LIN {X -0.159,Y -467.069,Z 497.488,A 0.000,B 0.000,C 90.000,E1 267.879} C_DIS
LIN {X -0.213,Y -463.902,Z 497.487,A 0.000,B 0.000,C 90.000,E1 267.650} C_DIS
LIN {X 0.193,Y -457.241,Z 497.485,A 0.000,B 0.000,C 90.000,E1 267.192} C_DIS
LIN {X -0.207,Y -450.486,Z 497.483,A 0.000,B 0.000,C 90.000,E1 266.906} C_DIS
LIN {X -0.134,Y -443.636,Z 497.481,A 0.000,B 0.000,C 90.000,E1 266.617} C_DIS
LIN {X -0.213,Y -436.403,Z 497.480,A 0.000,B 0.000,C 90.000,E1 266.388} C_DIS
LIN {X 0.056,Y -428.030,Z 497.479,A 0.000,B 0.000,C 90.000,E1 266.159} C_DIS
LIN {X -0.086,Y -418.559,Z 497.478,A 0.000,B 0.000,C 90.000,E1 266.045} C_DIS
LIN {X -0.068,Y -410.848,Z 497.478,A 0.000,B 0.000,C 90.000,E1 265.988} C_DIS
LIN {X -0.145,Y -404.938,Z 497.478,A 0.000,B 0.000,C 90.000,E1 265.988} C_DIS
LIN {X 0.081,Y -180.918,Z 497.478,A 0.000,B 0.000,C 90.000,E1 265.931} C_DIS
LIN {X -0.058,Y -180.845,Z 497.472,A 0.000,B 0.000,C 90.000,E1 264.951} C_DIS
LIN {X 0.019,Y -178.890,Z 497.443,A 0.000,B 0.000,C 90.000,E1 259.690} C_DIS
LIN {X -0.077,Y -175.932,Z 497.414,A 0.000,B 0.000,C 90.000,E1 254.629} C_DIS
LIN {X 0.040,Y -175.379,Z 497.410,A 0.000,B 0.000,C 90.000,E1 253.740} C_DIS
LIN {X 0.037,Y -172.153,Z 497.386,A 0.000,B 0.000,C 90.000,E1 249.464} C_DIS
LIN {X 0.074,Y -171.618,Z 497.381,A 0.000,B 0.000,C 90.000,E1 248.592} C_DIS
LIN {X 0.062,Y -167.841,Z 497.357,A 0.000,B 0.000,C 90.000,E1 244.280} C_DIS
LIN {X 0.002,Y -166.570,Z 497.348,A 0.000,B 0.000,C 90.000,E1 242.564} C_DIS
LIN {X -0.012,Y -162.563,Z 497.323,A 0.000,B 0.000,C 90.000,E1 238.201} C_DIS
LIN {X 0.048,Y -161.244,Z 497.314,A 0.000,B 0.000,C 90.000,E1 236.421} C_DIS
LIN {X -0.041,Y -157.247,Z 497.289,A 0.000,B 0.000,C 90.000,E1 232.029} C_DIS
LIN {X 0.005,Y -155.969,Z 497.279,A 0.000,B 0.000,C 90.000,E1 230.231} C_DIS
LIN {X 0.063,Y -152.224,Z 497.254,A 0.000,B 0.000,C 90.000,E1 225.729} C_DIS
LIN {X -0.027,Y -150.467,Z 497.239,A 0.000,B 0.000,C 90.000,E1 223.056} C_DIS
LIN {X -0.006,Y -147.192,Z 497.214,A 0.000,B 0.000,C 90.000,E1 218.508} C_DIS
LIN {X 0.076,Y -145.211,Z 497.194,A 0.000,B 0.000,C 90.000,E1 214.818} C_DIS
LIN {X -0.015,Y -142.344,Z 497.163,A 0.000,B 0.000,C 90.000,E1 209.333} C_DIS
LIN {X 0.039,Y -141.732,Z 497.153,A 0.000,B 0.000,C 90.000,E1 207.462} C_DIS
LIN {X 0.020,Y -139.483,Z 497.117,A 0.000,B 0.000,C 90.000,E1 200.972} C_DIS
LIN {X 0.009,Y -138.982,Z 497.101,A 0.000,B 0.000,C 90.000,E1 198.181} C_DIS
LIN {X -0.030,Y -138.333,Z 497.054,A 0.000,B 0.000,C 90.000,E1 189.792} C_DIS
LIN {X -0.006,Y -139.426,Z 497.008,A 0.000,B 0.000,C 90.000,E1 181.375} C_DIS
LIN {X 0.048,Y -141.349,Z 496.971,A 0.000,B 0.000,C 90.000,E1 174.837} C_DIS
LIN {X 0.025,Y -142.704,Z 496.956,A 0.000,B 0.000,C 90.000,E1 172.064} C_DIS
LIN {X -0.017,Y -145.075,Z 496.930,A 0.000,B 0.000,C 90.000,E1 167.465} C_DIS
LIN {X -0.020,Y -147.700,Z 496.910,A 0.000,B 0.000,C 90.000,E1 163.795} C_DIS
LIN {X 0.013,Y -150.352,Z 496.890,A 0.000,B 0.000,C 90.000,E1 160.134} C_DIS
LIN {X 0.005,Y -154.606,Z 496.865,A 0.000,B 0.000,C 90.000,E1 155.613} C_DIS
LIN {X 0.012,Y -158.148,Z 496.845,A 0.000,B 0.000,C 90.000,E1 152.025} C_DIS
LIN {X 0.057,Y -162.434,Z 496.825,A 0.000,B 0.000,C 90.000,E1 148.456} C_DIS
LIN {X -0.048,Y -166.694,Z 496.805,A 0.000,B 0.000,C 90.000,E1 144.975} C_DIS
LIN {X 0.066,Y -171.699,Z 496.786,A 0.000,B 0.000,C 90.000,E1 141.457} C_DIS
LIN {X 0.001,Y -176.673,Z 496.767,A 0.000,B 0.000,C 90.000,E1 138.038} C_DIS
LIN {X -0.006,Y -180.969,Z 496.753,A 0.000,B 0.000,C 90.000,E1 135.486} C_DIS
LIN {X -0.018,Y -186.393,Z 496.734,A 0.000,B 0.000,C 90.000,E1 132.123} C_DIS
LIN {X -0.078,Y -191.022,Z 496.720,A 0.000,B 0.000,C 90.000,E1 129.644} C_DIS
LIN {X -0.011,Y -192.947,Z 496.714,A 0.000,B 0.000,C 90.000,E1 128.463} C_DIS
LIN {X -0.063,Y -289.891,Z 496.714,A 0.000,B 0.000,C 90.000,E1 128.463} C_DIS
LIN {X -0.037,Y -294.322,Z 496.713,A 0.000,B 0.000,C 90.000,E1 128.338} C_DIS
LIN {X -0.058,Y -296.327,Z 496.712,A 0.000,B 0.000,C 90.000,E1 128.222} C_DIS
LIN {X -0.001,Y -299.079,Z 496.711,A 0.000,B 0.000,C 90.000,E1 127.971} C_DIS
LIN {X 0.099,Y -302.846,Z 496.708,A 0.000,B 0.000,C 90.000,E1 127.443} C_DIS
LIN {X -0.139,Y -304.561,Z 496.706,A 0.000,B 0.000,C 90.000,E1 127.156} C_DIS
LIN {X 0.049,Y -305.909,Z 496.704,A 0.000,B 0.000,C 90.000,E1 126.790} C_DIS
LIN {X 0.014,Y -317.009,Z 496.685,A 0.000,B 0.000,C 90.000,E1 123.214} C_DIS
LIN {X 0.034,Y -327.372,Z 496.669,A 0.000,B 0.000,C 90.000,E1 120.335} C_DIS
LIN {X 0.035,Y -339.088,Z 496.653,A 0.000,B 0.000,C 90.000,E1 117.513} C_DIS
LIN {X -0.109,Y -352.268,Z 496.638,A 0.000,B 0.000,C 90.000,E1 114.771} C_DIS
LIN {X 0.090,Y -365.305,Z 496.624,A 0.000,B 0.000,C 90.000,E1 112.333} C_DIS
LIN {X 0.000,Y -379.685,Z 496.611,A 0.000,B 0.000,C 90.000,E1 109.993} C_DIS
LIN {X 0.004,Y -395.513,Z 496.598,A 0.000,B 0.000,C 90.000,E1 107.692} C_DIS
LIN {X 0.171,Y -412.905,Z 496.586,A 0.000,B 0.000,C 90.000,E1 105.426} C_DIS
LIN {X 0.169,Y -431.991,Z 496.574,A 0.000,B 0.000,C 90.000,E1 103.244} C_DIS
LIN {X -0.185,Y -452.129,Z 496.562,A 0.000,B 0.000,C 90.000,E1 101.243} C_DIS
LIN {X 0.176,Y -472.814,Z 496.552,A 0.000,B 0.000,C 90.000,E1 99.321} C_DIS
LIN {X -0.004,Y -480.554,Z 496.548,A 0.000,B 0.000,C 90.000,E1 98.681} C_DIS
LIN {X 0.071,Y -482.476,Z 496.547,A 0.000,B 0.000,C 90.000,E1 98.454} C_DIS
LIN {X -0.051,Y -484.150,Z 496.546,A 0.000,B 0.000,C 90.000,E1 98.219} C_DIS
LIN {X -0.242,Y -485.406,Z 496.544,A 0.000,B 0.000,C 90.000,E1 97.992} C_DIS
LIN {X 0.010,Y -486.954,Z 496.541,A 0.000,B 0.000,C 90.000,E1 97.466} C_DIS
LIN {X 0.203,Y -487.446,Z 496.539,A 0.000,B 0.000,C 90.000,E1 96.947} C_DIS
LIN {X -0.078,Y -486.959,Z 496.536,A 0.000,B 0.000,C 90.000,E1 96.486} C_DIS
LIN {X 0.128,Y -485.415,Z 496.533,A 0.000,B 0.000,C 90.000,E1 95.967} C_DIS
LIN {X -0.037,Y -484.162,Z 496.532,A 0.000,B 0.000,C 90.000,E1 95.739} C_DIS
LIN {X -0.199,Y -482.489,Z 496.530,A 0.000,B 0.000,C 90.000,E1 95.511} C_DIS
LIN {X 0.089,Y -468.245,Z 496.521,A 0.000,B 0.000,C 90.000,E1 93.726} C_DIS
LIN {X 0.037,Y -455.064,Z 496.511,A 0.000,B 0.000,C 90.000,E1 91.949} C_DIS
LIN {X 0.020,Y -436.764,Z 496.495,A 0.000,B 0.000,C 90.000,E1 89.083} C_DIS
LIN {X -0.075,Y -423.680,Z 496.483,A 0.000,B 0.000,C 90.000,E1 86.963} C_DIS
LIN {X -0.085,Y -412.501,Z 496.473,A 0.000,B 0.000,C 90.000,E1 85.065} C_DIS
LIN {X -0.194,Y -398.290,Z 496.459,A 0.000,B 0.000,C 90.000,E1 82.591} C_DIS
LIN {X 0.156,Y -387.289,Z 496.448,A 0.000,B 0.000,C 90.000,E1 80.566} C_DIS
LIN {X 0.036,Y -374.741,Z 496.435,A 0.000,B 0.000,C 90.000,E1 78.285} C_DIS
LIN {X 0.008,Y -359.680,Z 496.419,A 0.000,B 0.000,C 90.000,E1 75.353} C_DIS
LIN {X -0.041,Y -349.044,Z 496.405,A 0.000,B 0.000,C 90.000,E1 72.960} C_DIS
LIN {X 0.086,Y -335.271,Z 496.385,A 0.000,B 0.000,C 90.000,E1 69.263} C_DIS
LIN {X -0.128,Y -324.859,Z 496.368,A 0.000,B 0.000,C 90.000,E1 66.177} C_DIS
LIN {X -0.128,Y -316.777,Z 496.353,A 0.000,B 0.000,C 90.000,E1 63.640} C_DIS
LIN {X -0.043,Y -308.825,Z 496.339,A 0.000,B 0.000,C 90.000,E1 61.051} C_DIS
LIN {X -0.122,Y -300.916,Z 496.325,A 0.000,B 0.000,C 90.000,E1 58.456} C_DIS
LIN {X 0.082,Y -291.407,Z 496.306,A 0.000,B 0.000,C 90.000,E1 55.102} C_DIS
LIN {X -0.032,Y -284.211,Z 496.291,A 0.000,B 0.000,C 90.000,E1 52.431} C_DIS
LIN {X 0.125,Y -278.713,Z 496.280,A 0.000,B 0.000,C 90.000,E1 50.356} C_DIS
LIN {X -0.028,Y -274.824,Z 496.272,A 0.000,B 0.000,C 90.000,E1 49.013} C_DIS
LIN {X -0.048,Y -270.703,Z 496.265,A 0.000,B 0.000,C 90.000,E1 47.634} C_DIS
LIN {X 0.005,Y -264.053,Z 496.253,A 0.000,B 0.000,C 90.000,E1 45.526} C_DIS
LIN {X -0.062,Y -255.999,Z 496.239,A 0.000,B 0.000,C 90.000,E1 43.056} C_DIS
LIN {X -0.069,Y -245.974,Z 496.221,A 0.000,B 0.000,C 90.000,E1 39.806} C_DIS
LIN {X 0.062,Y -235.445,Z 496.201,A 0.000,B 0.000,C 90.000,E1 36.091} C_DIS
LIN {X 0.070,Y -227.752,Z 496.184,A 0.000,B 0.000,C 90.000,E1 33.086} C_DIS
LIN {X 0.016,Y -221.019,Z 496.167,A 0.000,B 0.000,C 90.000,E1 30.050} C_DIS
LIN {X 0.048,Y -215.087,Z 496.150,A 0.000,B 0.000,C 90.000,E1 26.950} C_DIS
LIN {X 0.033,Y -210.049,Z 496.132,A 0.000,B 0.000,C 90.000,E1 23.823} C_DIS
LIN {X -0.045,Y -204.859,Z 496.110,A 0.000,B 0.000,C 90.000,E1 19.885} C_DIS
LIN {X 0.094,Y -200.523,Z 496.088,A 0.000,B 0.000,C 90.000,E1 15.843} C_DIS
LIN {X 0.044,Y -196.735,Z 496.061,A 0.000,B 0.000,C 90.000,E1 11.007} C_DIS
LIN {X 0.081,Y -193.879,Z 496.025,A 0.000,B 0.000,C 90.000,E1 4.473} C_DIS
LIN {X -0.057,Y -194.901,Z 495.961,A 0.000,B 0.000,C 90.000,E1 352.996} C_DIS
LIN {X -0.067,Y -197.808,Z 495.934,A 0.000,B 0.000,C 90.000,E1 348.105} C_DIS
LIN {X 0.014,Y -201.345,Z 495.911,A 0.000,B 0.000,C 90.000,E1 344.031} C_DIS
LIN {X 0.035,Y -205.757,Z 495.889,A 0.000,B 0.000,C 90.000,E1 340.007} C_DIS
LIN {X -0.038,Y -211.033,Z 495.867,A 0.000,B 0.000,C 90.000,E1 336.049} C_DIS
LIN {X 0.016,Y -216.916,Z 495.845,A 0.000,B 0.000,C 90.000,E1 332.103} C_DIS
LIN {X 0.093,Y -223.417,Z 495.823,A 0.000,B 0.000,C 90.000,E1 328.201} C_DIS
LIN {X -0.023,Y -230.541,Z 495.802,A 0.000,B 0.000,C 90.000,E1 324.402} C_DIS
LIN {X -0.069,Y -238.308,Z 495.781,A 0.000,B 0.000,C 90.000,E1 320.642} C_DIS
LIN {X 0.042,Y -247.097,Z 495.761,A 0.000,B 0.000,C 90.000,E1 316.905} C_DIS
LIN {X 0.028,Y -253.961,Z 495.746,A 0.000,B 0.000,C 90.000,E1 314.352} C_DIS
LIN {X -0.044,Y -264.868,Z 495.727,A 0.000,B 0.000,C 90.000,E1 310.782} C_DIS
LIN {X 0.031,Y -275.649,Z 495.709,A 0.000,B 0.000,C 90.000,E1 307.604} C_DIS
LIN {X -0.123,Y -288.837,Z 495.690,A 0.000,B 0.000,C 90.000,E1 304.199} C_DIS
LIN {X 0.128,Y -301.582,Z 495.673,A 0.000,B 0.000,C 90.000,E1 301.131} C_DIS
LIN {X -0.084,Y -316.818,Z 495.655,A 0.000,B 0.000,C 90.000,E1 297.897} C_DIS
LIN {X -0.042,Y -330.447,Z 495.641,A 0.000,B 0.000,C 90.000,E1 295.335} C_DIS
LIN {X 0.069,Y -343.666,Z 495.629,A 0.000,B 0.000,C 90.000,E1 293.131} C_DIS
LIN {X 0.220,Y -358.136,Z 495.617,A 0.000,B 0.000,C 90.000,E1 290.972} C_DIS
LIN {X 0.100,Y -373.737,Z 495.605,A 0.000,B 0.000,C 90.000,E1 288.906} C_DIS
LIN {X -0.133,Y -393.034,Z 495.592,A 0.000,B 0.000,C 90.000,E1 286.622} C_DIS
LIN {X -0.119,Y -415.555,Z 495.578,A 0.000,B 0.000,C 90.000,E1 284.120} C_DIS
LIN {X -0.049,Y -428.141,Z 495.571,A 0.000,B 0.000,C 90.000,E1 282.771} C_DIS
LIN {X 0.056,Y -440.413,Z 495.564,A 0.000,B 0.000,C 90.000,E1 281.422} C_DIS
LIN {X 0.058,Y -449.879,Z 495.558,A 0.000,B 0.000,C 90.000,E1 280.366} C_DIS
LIN {X -0.177,Y -456.408,Z 495.553,A 0.000,B 0.000,C 90.000,E1 279.613} C_DIS
LIN {X 0.106,Y -462.355,Z 495.549,A 0.000,B 0.000,C 90.000,E1 278.803} C_DIS
LIN {X -0.018,Y -467.762,Z 495.545,A 0.000,B 0.000,C 90.000,E1 278.049} C_DIS
LIN {X -0.092,Y -472.644,Z 495.540,A 0.000,B 0.000,C 90.000,E1 277.296} C_DIS
LIN {X -0.133,Y -476.909,Z 495.536,A 0.000,B 0.000,C 90.000,E1 276.543} C_DIS
LIN {X -0.187,Y -480.642,Z 495.532,A 0.000,B 0.000,C 90.000,E1 275.796} C_DIS
LIN {X -0.209,Y -483.765,Z 495.528,A 0.000,B 0.000,C 90.000,E1 275.049} C_DIS
LIN {X -0.037,Y -485.507,Z 495.525,A 0.000,B 0.000,C 90.000,E1 274.531} C_DIS
LIN {X 0.145,Y -486.903,Z 495.522,A 0.000,B 0.000,C 90.000,E1 274.012} C_DIS
LIN {X -0.182,Y -487.979,Z 495.520,A 0.000,B 0.000,C 90.000,E1 273.555} C_DIS
LIN {X 0.016,Y -488.764,Z 495.517,A 0.000,B 0.000,C 90.000,E1 273.037} C_DIS
LIN {X 0.194,Y -489.189,Z 495.514,A 0.000,B 0.000,C 90.000,E1 272.522} C_DIS
LIN {X -0.109,Y -489.235,Z 495.511,A 0.000,B 0.000,C 90.000,E1 272.064} C_DIS
LIN {X 0.095,Y -488.877,Z 495.509,A 0.000,B 0.000,C 90.000,E1 271.547} C_DIS
LIN {X -0.204,Y -488.107,Z 495.506,A 0.000,B 0.000,C 90.000,E1 271.088} C_DIS
LIN {X -0.016,Y -486.833,Z 495.503,A 0.000,B 0.000,C 90.000,E1 270.573} C_DIS
LIN {X 0.167,Y -485.001,Z 495.500,A 0.000,B 0.000,C 90.000,E1 270.057} C_DIS
LIN {X -0.141,Y -482.512,Z 495.498,A 0.000,B 0.000,C 90.000,E1 269.599} C_DIS
LIN {X 0.017,Y -479.232,Z 495.495,A 0.000,B 0.000,C 90.000,E1 269.083} C_DIS
LIN {X 0.155,Y -475.095,Z 495.492,A 0.000,B 0.000,C 90.000,E1 268.568} C_DIS
LIN {X -0.025,Y -472.680,Z 495.491,A 0.000,B 0.000,C 90.000,E1 268.339} C_DIS
LIN {X -0.224,Y -467.092,Z 495.488,A 0.000,B 0.000,C 90.000,E1 267.879} C_DIS
LIN {X -0.049,Y -460.845,Z 495.486,A 0.000,B 0.000,C 90.000,E1 267.421} C_DIS
LIN {X 0.179,Y -454.124,Z 495.484,A 0.000,B 0.000,C 90.000,E1 267.020} C_DIS
LIN {X 0.007,Y -447.262,Z 495.482,A 0.000,B 0.000,C 90.000,E1 266.731} C_DIS
LIN {X 0.211,Y -440.273,Z 495.480,A 0.000,B 0.000,C 90.000,E1 266.445} C_DIS
LIN {X -0.102,Y -432.652,Z 495.479,A 0.000,B 0.000,C 90.000,E1 266.274} C_DIS
LIN {X -0.021,Y -424.203,Z 495.478,A 0.000,B 0.000,C 90.000,E1 266.102} C_DIS
LIN {X 0.001,Y -413.442,Z 495.478,A 0.000,B 0.000,C 90.000,E1 265.988} C_DIS
LIN {X -0.161,Y -406.443,Z 495.478,A 0.000,B 0.000,C 90.000,E1 265.988} C_DIS
LIN {X 0.073,Y -180.918,Z 495.478,A 0.000,B 0.000,C 90.000,E1 265.931} C_DIS
LIN {X -0.068,Y -180.845,Z 495.472,A 0.000,B 0.000,C 90.000,E1 264.951} C_DIS
LIN {X 0.008,Y -178.889,Z 495.443,A 0.000,B 0.000,C 90.000,E1 259.690} C_DIS
LIN {X 0.083,Y -175.931,Z 495.414,A 0.000,B 0.000,C 90.000,E1 254.574} C_DIS
LIN {X 0.029,Y -175.376,Z 495.410,A 0.000,B 0.000,C 90.000,E1 253.740} C_DIS
LIN {X 0.027,Y -172.151,Z 495.386,A 0.000,B 0.000,C 90.000,E1 249.464} C_DIS
LIN {X 0.065,Y -171.617,Z 495.381,A 0.000,B 0.000,C 90.000,E1 248.592} C_DIS
LIN {X 0.053,Y -167.839,Z 495.357,A 0.000,B 0.000,C 90.000,E1 244.280} C_DIS
LIN {X -0.007,Y -166.567,Z 495.348,A 0.000,B 0.000,C 90.000,E1 242.564} C_DIS
LIN {X -0.020,Y -162.561,Z 495.323,A 0.000,B 0.000,C 90.000,E1 238.201} C_DIS
LIN {X 0.039,Y -161.240,Z 495.314,A 0.000,B 0.000,C 90.000,E1 236.421} C_DIS
LIN {X 0.074,Y -157.244,Z 495.289,A 0.000,B 0.000,C 90.000,E1 231.984} C_DIS
LIN {X -0.004,Y -155.967,Z 495.279,A 0.000,B 0.000,C 90.000,E1 230.231} C_DIS
LIN {X 0.054,Y -152.222,Z 495.254,A 0.000,B 0.000,C 90.000,E1 225.729} C_DIS
LIN {X -0.035,Y -150.465,Z 495.239,A 0.000,B 0.000,C 90.000,E1 223.056} C_DIS
LIN {X -0.015,Y -147.190,Z 495.214,A 0.000,B 0.000,C 90.000,E1 218.508} C_DIS
LIN {X 0.067,Y -145.209,Z 495.194,A 0.000,B 0.000,C 90.000,E1 214.818} C_DIS
LIN {X -0.023,Y -142.343,Z 495.163,A 0.000,B 0.000,C 90.000,E1 209.333} C_DIS
LIN {X 0.030,Y -141.731,Z 495.153,A 0.000,B 0.000,C 90.000,E1 207.462} C_DIS
LIN {X 0.012,Y -139.483,Z 495.117,A 0.000,B 0.000,C 90.000,E1 200.972} C_DIS
LIN {X 0.000,Y -138.982,Z 495.101,A 0.000,B 0.000,C 90.000,E1 198.181} C_DIS
LIN {X -0.038,Y -138.333,Z 495.054,A 0.000,B 0.000,C 90.000,E1 189.792} C_DIS
LIN {X -0.014,Y -139.427,Z 495.008,A 0.000,B 0.000,C 90.000,E1 181.375} C_DIS
LIN {X 0.040,Y -141.351,Z 494.971,A 0.000,B 0.000,C 90.000,E1 174.837} C_DIS
LIN {X 0.016,Y -142.705,Z 494.956,A 0.000,B 0.000,C 90.000,E1 172.064} C_DIS
LIN {X -0.025,Y -145.077,Z 494.930,A 0.000,B 0.000,C 90.000,E1 167.465} C_DIS
LIN {X -0.029,Y -147.702,Z 494.910,A 0.000,B 0.000,C 90.000,E1 163.795} C_DIS
LIN {X 0.054,Y -150.355,Z 494.890,A 0.000,B 0.000,C 90.000,E1 160.115} C_DIS
LIN {X 0.073,Y -153.779,Z 494.870,A 0.000,B 0.000,C 90.000,E1 156.485} C_DIS
LIN {X -0.007,Y -157.191,Z 494.850,A 0.000,B 0.000,C 90.000,E1 152.922} C_DIS
LIN {X 0.076,Y -161.351,Z 494.830,A 0.000,B 0.000,C 90.000,E1 149.331} C_DIS
LIN {X 0.088,Y -165.554,Z 494.810,A 0.000,B 0.000,C 90.000,E1 145.801} C_DIS
LIN {X -0.028,Y -170.468,Z 494.791,A 0.000,B 0.000,C 90.000,E1 142.351} C_DIS
LIN {X -0.011,Y -175.350,Z 494.772,A 0.000,B 0.000,C 90.000,E1 138.895} C_DIS
LIN {X -0.015,Y -180.974,Z 494.753,A 0.000,B 0.000,C 90.000,E1 135.486} C_DIS
LIN {X -0.028,Y -186.398,Z 494.734,A 0.000,B 0.000,C 90.000,E1 132.123} C_DIS
LIN {X -0.088,Y -191.027,Z 494.720,A 0.000,B 0.000,C 90.000,E1 129.644} C_DIS
LIN {X 0.094,Y -193.031,Z 494.713,A 0.000,B 0.000,C 90.000,E1 128.382} C_DIS
LIN {X 0.097,Y -290.712,Z 494.713,A 0.000,B 0.000,C 90.000,E1 128.382} C_DIS
LIN {X 0.009,Y -291.718,Z 494.713,A 0.000,B 0.000,C 90.000,E1 128.382} C_DIS
LIN {X -0.005,Y -296.314,Z 494.712,A 0.000,B 0.000,C 90.000,E1 128.177} C_DIS
LIN {X -0.017,Y -298.790,Z 494.711,A 0.000,B 0.000,C 90.000,E1 127.971} C_DIS
LIN {X 0.163,Y -302.616,Z 494.708,A 0.000,B 0.000,C 90.000,E1 127.443} C_DIS
LIN {X -0.075,Y -304.406,Z 494.706,A 0.000,B 0.000,C 90.000,E1 127.156} C_DIS
LIN {X 0.111,Y -305.809,Z 494.704,A 0.000,B 0.000,C 90.000,E1 126.790} C_DIS
LIN {X -0.089,Y -307.846,Z 494.701,A 0.000,B 0.000,C 90.000,E1 126.171} C_DIS
LIN {X 0.148,Y -318.034,Z 494.683,A 0.000,B 0.000,C 90.000,E1 122.880} C_DIS
LIN {X -0.076,Y -328.534,Z 494.667,A 0.000,B 0.000,C 90.000,E1 120.050} C_DIS
LIN {X 0.086,Y -340.403,Z 494.651,A 0.000,B 0.000,C 90.000,E1 117.206} C_DIS
LIN {X -0.006,Y -353.742,Z 494.636,A 0.000,B 0.000,C 90.000,E1 114.463} C_DIS
LIN {X -0.103,Y -366.936,Z 494.623,A 0.000,B 0.000,C 90.000,E1 112.078} C_DIS
LIN {X 0.065,Y -381.483,Z 494.610,A 0.000,B 0.000,C 90.000,E1 109.704} C_DIS
LIN {X 0.127,Y -397.492,Z 494.597,A 0.000,B 0.000,C 90.000,E1 107.402} C_DIS
LIN {X -0.040,Y -415.080,Z 494.584,A 0.000,B 0.000,C 90.000,E1 105.190} C_DIS
LIN {X 0.030,Y -434.343,Z 494.572,A 0.000,B 0.000,C 90.000,E1 103.008} C_DIS
LIN {X -0.167,Y -454.551,Z 494.561,A 0.000,B 0.000,C 90.000,E1 101.007} C_DIS
LIN {X -0.193,Y -475.297,Z 494.551,A 0.000,B 0.000,C 90.000,E1 99.151} C_DIS
LIN {X 0.060,Y -480.475,Z 494.548,A 0.000,B 0.000,C 90.000,E1 98.681} C_DIS
LIN {X 0.135,Y -482.460,Z 494.547,A 0.000,B 0.000,C 90.000,E1 98.454} C_DIS
LIN {X 0.013,Y -484.182,Z 494.546,A 0.000,B 0.000,C 90.000,E1 98.219} C_DIS
LIN {X -0.178,Y -485.476,Z 494.544,A 0.000,B 0.000,C 90.000,E1 97.992} C_DIS
LIN {X 0.074,Y -487.079,Z 494.542,A 0.000,B 0.000,C 90.000,E1 97.466} C_DIS
LIN {X -0.216,Y -487.616,Z 494.539,A 0.000,B 0.000,C 90.000,E1 97.004} C_DIS
LIN {X -0.013,Y -487.173,Z 494.536,A 0.000,B 0.000,C 90.000,E1 96.486} C_DIS
LIN {X 0.193,Y -485.682,Z 494.533,A 0.000,B 0.000,C 90.000,E1 95.967} C_DIS
LIN {X 0.030,Y -484.462,Z 494.532,A 0.000,B 0.000,C 90.000,E1 95.739} C_DIS
LIN {X -0.132,Y -482.833,Z 494.531,A 0.000,B 0.000,C 90.000,E1 95.511} C_DIS
LIN {X -0.114,Y -470.618,Z 494.522,A 0.000,B 0.000,C 90.000,E1 94.012} C_DIS
LIN {X -0.125,Y -457.192,Z 494.512,A 0.000,B 0.000,C 90.000,E1 92.236} C_DIS
LIN {X 0.066,Y -445.210,Z 494.502,A 0.000,B 0.000,C 90.000,E1 90.401} C_DIS
LIN {X -0.002,Y -433.770,Z 494.492,A 0.000,B 0.000,C 90.000,E1 88.568} C_DIS
LIN {X 0.100,Y -417.547,Z 494.477,A 0.000,B 0.000,C 90.000,E1 85.869} C_DIS
LIN {X 0.028,Y -404.810,Z 494.465,A 0.000,B 0.000,C 90.000,E1 83.685} C_DIS
LIN {X 0.074,Y -393.852,Z 494.454,A 0.000,B 0.000,C 90.000,E1 81.724} C_DIS
LIN {X 0.002,Y -382.829,Z 494.443,A 0.000,B 0.000,C 90.000,E1 79.746} C_DIS
LIN {X 0.152,Y -370.337,Z 494.430,A 0.000,B 0.000,C 90.000,E1 77.409} C_DIS
LIN {X 0.111,Y -359.905,Z 494.419,A 0.000,B 0.000,C 90.000,E1 75.353} C_DIS
LIN {X -0.013,Y -348.012,Z 494.404,A 0.000,B 0.000,C 90.000,E1 72.670} C_DIS
LIN {X 0.193,Y -335.424,Z 494.385,A 0.000,B 0.000,C 90.000,E1 69.263} C_DIS
LIN {X -0.020,Y -324.965,Z 494.368,A 0.000,B 0.000,C 90.000,E1 66.177} C_DIS
LIN {X -0.020,Y -316.855,Z 494.354,A 0.000,B 0.000,C 90.000,E1 63.640} C_DIS
LIN {X 0.064,Y -308.873,Z 494.339,A 0.000,B 0.000,C 90.000,E1 61.051} C_DIS
LIN {X -0.017,Y -300.929,Z 494.325,A 0.000,B 0.000,C 90.000,E1 58.456} C_DIS
LIN {X 0.018,Y -291.391,Z 494.306,A 0.000,B 0.000,C 90.000,E1 55.135} C_DIS
LIN {X 0.067,Y -284.165,Z 494.291,A 0.000,B 0.000,C 90.000,E1 52.431} C_DIS
LIN {X -0.171,Y -278.656,Z 494.280,A 0.000,B 0.000,C 90.000,E1 50.436} C_DIS
LIN {X 0.061,Y -272.726,Z 494.269,A 0.000,B 0.000,C 90.000,E1 48.324} C_DIS
LIN {X 0.013,Y -268.472,Z 494.261,A 0.000,B 0.000,C 90.000,E1 46.944} C_DIS
LIN {X 0.145,Y -262.873,Z 494.251,A 0.000,B 0.000,C 90.000,E1 45.162} C_DIS
LIN {X 0.060,Y -254.852,Z 494.237,A 0.000,B 0.000,C 90.000,E1 42.690} C_DIS
LIN {X 0.014,Y -245.992,Z 494.221,A 0.000,B 0.000,C 90.000,E1 39.806} C_DIS
LIN {X -0.048,Y -235.450,Z 494.201,A 0.000,B 0.000,C 90.000,E1 36.137} C_DIS
LIN {X 0.022,Y -227.743,Z 494.184,A 0.000,B 0.000,C 90.000,E1 33.118} C_DIS
LIN {X -0.020,Y -221.036,Z 494.167,A 0.000,B 0.000,C 90.000,E1 30.079} C_DIS
LIN {X -0.070,Y -215.102,Z 494.150,A 0.000,B 0.000,C 90.000,E1 27.001} C_DIS
LIN {X 0.105,Y -210.054,Z 494.133,A 0.000,B 0.000,C 90.000,E1 23.823} C_DIS
LIN {X 0.026,Y -204.841,Z 494.111,A 0.000,B 0.000,C 90.000,E1 19.885} C_DIS
LIN {X -0.030,Y -200.494,Z 494.088,A 0.000,B 0.000,C 90.000,E1 15.898} C_DIS
LIN {X 0.072,Y -196.682,Z 494.061,A 0.000,B 0.000,C 90.000,E1 11.018} C_DIS
LIN {X -0.050,Y -193.809,Z 494.025,A 0.000,B 0.000,C 90.000,E1 4.531} C_DIS
LIN {X -0.038,Y -194.787,Z 493.961,A 0.000,B 0.000,C 90.000,E1 352.989} C_DIS
LIN {X -0.076,Y -197.682,Z 493.934,A 0.000,B 0.000,C 90.000,E1 348.105} C_DIS
LIN {X 0.099,Y -202.038,Z 493.907,A 0.000,B 0.000,C 90.000,E1 343.196} C_DIS
LIN {X 0.013,Y -206.620,Z 493.885,A 0.000,B 0.000,C 90.000,E1 339.209} C_DIS
LIN {X 0.050,Y -212.019,Z 493.862,A 0.000,B 0.000,C 90.000,E1 335.229} C_DIS
LIN {X 0.044,Y -218.036,Z 493.841,A 0.000,B 0.000,C 90.000,E1 331.307} C_DIS
LIN {X -0.030,Y -224.656,Z 493.819,A 0.000,B 0.000,C 90.000,E1 327.454} C_DIS
LIN {X 0.021,Y -231.900,Z 493.798,A 0.000,B 0.000,C 90.000,E1 323.623} C_DIS
LIN {X 0.013,Y -239.859,Z 493.777,A 0.000,B 0.000,C 90.000,E1 319.865} C_DIS
LIN {X 0.151,Y -248.873,Z 493.757,A 0.000,B 0.000,C 90.000,E1 316.134} C_DIS
LIN {X 0.039,Y -258.169,Z 493.738,A 0.000,B 0.000,C 90.000,E1 312.894} C_DIS
LIN {X -0.053,Y -269.475,Z 493.719,A 0.000,B 0.000,C 90.000,E1 309.358} C_DIS
LIN {X -0.072,Y -282.107,Z 493.699,A 0.000,B 0.000,C 90.000,E1 305.884} C_DIS
LIN {X 0.047,Y -295.843,Z 493.680,A 0.000,B 0.000,C 90.000,E1 302.467} C_DIS
LIN {X 0.073,Y -310.559,Z 493.662,A 0.000,B 0.000,C 90.000,E1 299.155} C_DIS
LIN {X -0.107,Y -321.798,Z 493.649,A 0.000,B 0.000,C 90.000,E1 296.924} C_DIS
LIN {X -0.051,Y -334.118,Z 493.637,A 0.000,B 0.000,C 90.000,E1 294.695} C_DIS
LIN {X 0.022,Y -349.716,Z 493.623,A 0.000,B 0.000,C 90.000,E1 292.206} C_DIS
LIN {X -0.025,Y -369.142,Z 493.608,A 0.000,B 0.000,C 90.000,E1 289.504} C_DIS
LIN {X -0.014,Y -388.161,Z 493.595,A 0.000,B 0.000,C 90.000,E1 287.166} C_DIS
LIN {X 0.174,Y -412.902,Z 493.580,A 0.000,B 0.000,C 90.000,E1 284.356} C_DIS
LIN {X 0.070,Y -427.960,Z 493.571,A 0.000,B 0.000,C 90.000,E1 282.771} C_DIS
LIN {X -0.212,Y -440.245,Z 493.564,A 0.000,B 0.000,C 90.000,E1 281.478} C_DIS
LIN {X 0.223,Y -449.754,Z 493.558,A 0.000,B 0.000,C 90.000,E1 280.366} C_DIS
LIN {X -0.010,Y -456.319,Z 493.553,A 0.000,B 0.000,C 90.000,E1 279.613} C_DIS
LIN {X -0.183,Y -462.286,Z 493.549,A 0.000,B 0.000,C 90.000,E1 278.859} C_DIS
LIN {X -0.009,Y -469.446,Z 493.543,A 0.000,B 0.000,C 90.000,E1 277.814} C_DIS
LIN {X -0.135,Y -474.129,Z 493.539,A 0.000,B 0.000,C 90.000,E1 277.068} C_DIS
LIN {X -0.158,Y -478.241,Z 493.535,A 0.000,B 0.000,C 90.000,E1 276.315} C_DIS
LIN {X -0.202,Y -481.788,Z 493.531,A 0.000,B 0.000,C 90.000,E1 275.568} C_DIS
LIN {X -0.035,Y -483.823,Z 493.528,A 0.000,B 0.000,C 90.000,E1 275.049} C_DIS
LIN {X 0.138,Y -485.560,Z 493.525,A 0.000,B 0.000,C 90.000,E1 274.531} C_DIS
LIN {X -0.164,Y -486.996,Z 493.522,A 0.000,B 0.000,C 90.000,E1 274.069} C_DIS
LIN {X -0.005,Y -488.124,Z 493.520,A 0.000,B 0.000,C 90.000,E1 273.555} C_DIS
LIN {X 0.193,Y -488.894,Z 493.517,A 0.000,B 0.000,C 90.000,E1 273.037} C_DIS
LIN {X -0.116,Y -489.326,Z 493.514,A 0.000,B 0.000,C 90.000,E1 272.579} C_DIS
LIN {X 0.071,Y -489.410,Z 493.512,A 0.000,B 0.000,C 90.000,E1 272.064} C_DIS
LIN {X -0.213,Y -489.094,Z 493.509,A 0.000,B 0.000,C 90.000,E1 271.604} C_DIS
LIN {X -0.023,Y -488.341,Z 493.506,A 0.000,B 0.000,C 90.000,E1 271.088} C_DIS
LIN {X 0.166,Y -487.098,Z 493.503,A 0.000,B 0.000,C 90.000,E1 270.573} C_DIS
LIN {X -0.135,Y -485.245,Z 493.501,A 0.000,B 0.000,C 90.000,E1 270.115} C_DIS
LIN {X 0.042,Y -482.794,Z 493.498,A 0.000,B 0.000,C 90.000,E1 269.599} C_DIS
LIN {X 0.200,Y -479.589,Z 493.495,A 0.000,B 0.000,C 90.000,E1 269.083} C_DIS
LIN {X -0.137,Y -475.449,Z 493.492,A 0.000,B 0.000,C 90.000,E1 268.625} C_DIS
LIN {X 0.159,Y -473.063,Z 493.491,A 0.000,B 0.000,C 90.000,E1 268.339} C_DIS
LIN {X -0.041,Y -467.546,Z 493.488,A 0.000,B 0.000,C 90.000,E1 267.879} C_DIS
LIN {X 0.117,Y -461.350,Z 493.486,A 0.000,B 0.000,C 90.000,E1 267.421} C_DIS
LIN {X -0.146,Y -454.684,Z 493.484,A 0.000,B 0.000,C 90.000,E1 267.078} C_DIS
LIN {X 0.102,Y -447.788,Z 493.482,A 0.000,B 0.000,C 90.000,E1 266.731} C_DIS
LIN {X -0.148,Y -440.778,Z 493.480,A 0.000,B 0.000,C 90.000,E1 266.502} C_DIS
LIN {X -0.028,Y -433.298,Z 493.479,A 0.000,B 0.000,C 90.000,E1 266.274} C_DIS
LIN {X 0.030,Y -424.905,Z 493.478,A 0.000,B 0.000,C 90.000,E1 266.102} C_DIS
LIN {X 0.026,Y -414.498,Z 493.478,A 0.000,B 0.000,C 90.000,E1 265.988} C_DIS
LIN {X -0.180,Y -407.376,Z 493.478,A 0.000,B 0.000,C 90.000,E1 265.988} C_DIS
LIN {X 0.083,Y -180.918,Z 493.478,A 0.000,B 0.000,C 90.000,E1 265.931} C_DIS
LIN {X -0.059,Y -180.845,Z 493.472,A 0.000,B 0.000,C 90.000,E1 264.951} C_DIS
LIN {X 0.018,Y -178.889,Z 493.443,A 0.000,B 0.000,C 90.000,E1 259.690} C_DIS
LIN {X -0.077,Y -175.932,Z 493.414,A 0.000,B 0.000,C 90.000,E1 254.629} C_DIS
LIN {X 0.038,Y -175.378,Z 493.410,A 0.000,B 0.000,C 90.000,E1 253.740} C_DIS
LIN {X 0.035,Y -172.152,Z 493.386,A 0.000,B 0.000,C 90.000,E1 249.464} C_DIS
LIN {X 0.073,Y -171.619,Z 493.381,A 0.000,B 0.000,C 90.000,E1 248.592} C_DIS
LIN {X 0.062,Y -167.841,Z 493.357,A 0.000,B 0.000,C 90.000,E1 244.280} C_DIS
LIN {X 0.001,Y -166.570,Z 493.348,A 0.000,B 0.000,C 90.000,E1 242.564} C_DIS
LIN {X -0.012,Y -162.563,Z 493.323,A 0.000,B 0.000,C 90.000,E1 238.201} C_DIS
LIN {X 0.048,Y -161.243,Z 493.314,A 0.000,B 0.000,C 90.000,E1 236.421} C_DIS
LIN {X -0.042,Y -157.247,Z 493.289,A 0.000,B 0.000,C 90.000,E1 232.029} C_DIS
LIN {X 0.005,Y -155.970,Z 493.279,A 0.000,B 0.000,C 90.000,E1 230.231} C_DIS
LIN {X 0.063,Y -152.224,Z 493.254,A 0.000,B 0.000,C 90.000,E1 225.729} C_DIS
LIN {X -0.027,Y -150.467,Z 493.239,A 0.000,B 0.000,C 90.000,E1 223.056} C_DIS
LIN {X -0.006,Y -147.192,Z 493.214,A 0.000,B 0.000,C 90.000,E1 218.508} C_DIS
LIN {X 0.074,Y -145.211,Z 493.194,A 0.000,B 0.000,C 90.000,E1 214.818} C_DIS
LIN {X -0.015,Y -142.343,Z 493.163,A 0.000,B 0.000,C 90.000,E1 209.333} C_DIS
LIN {X 0.037,Y -141.732,Z 493.153,A 0.000,B 0.000,C 90.000,E1 207.462} C_DIS
LIN {X 0.019,Y -139.483,Z 493.117,A 0.000,B 0.000,C 90.000,E1 200.972} C_DIS
LIN {X 0.008,Y -138.983,Z 493.101,A 0.000,B 0.000,C 90.000,E1 198.181} C_DIS
LIN {X -0.030,Y -138.333,Z 493.054,A 0.000,B 0.000,C 90.000,E1 189.792} C_DIS
LIN {X -0.006,Y -139.426,Z 493.008,A 0.000,B 0.000,C 90.000,E1 181.375} C_DIS
LIN {X 0.048,Y -141.349,Z 492.971,A 0.000,B 0.000,C 90.000,E1 174.837} C_DIS
LIN {X 0.024,Y -142.704,Z 492.956,A 0.000,B 0.000,C 90.000,E1 172.064} C_DIS
LIN {X -0.017,Y -145.076,Z 492.930,A 0.000,B 0.000,C 90.000,E1 167.465} C_DIS
LIN {X -0.021,Y -147.700,Z 492.910,A 0.000,B 0.000,C 90.000,E1 163.795} C_DIS
LIN {X 0.012,Y -150.352,Z 492.890,A 0.000,B 0.000,C 90.000,E1 160.134} C_DIS
LIN {X 0.005,Y -154.606,Z 492.865,A 0.000,B 0.000,C 90.000,E1 155.613} C_DIS
LIN {X 0.012,Y -158.148,Z 492.845,A 0.000,B 0.000,C 90.000,E1 152.025} C_DIS
LIN {X 0.056,Y -162.435,Z 492.825,A 0.000,B 0.000,C 90.000,E1 148.456} C_DIS
LIN {X -0.048,Y -166.694,Z 492.805,A 0.000,B 0.000,C 90.000,E1 144.975} C_DIS
LIN {X 0.065,Y -171.700,Z 492.786,A 0.000,B 0.000,C 90.000,E1 141.457} C_DIS
LIN {X -0.001,Y -176.673,Z 492.767,A 0.000,B 0.000,C 90.000,E1 138.038} C_DIS
LIN {X -0.006,Y -180.969,Z 492.753,A 0.000,B 0.000,C 90.000,E1 135.486} C_DIS
LIN {X -0.019,Y -186.394,Z 492.734,A 0.000,B 0.000,C 90.000,E1 132.123} C_DIS
LIN {X -0.079,Y -191.023,Z 492.720,A 0.000,B 0.000,C 90.000,E1 129.644} C_DIS
LIN {X -0.034,Y -193.097,Z 492.713,A 0.000,B 0.000,C 90.000,E1 128.382} C_DIS
LIN {X -0.086,Y -289.820,Z 492.713,A 0.000,B 0.000,C 90.000,E1 128.382} C_DIS
LIN {X -0.033,Y -292.205,Z 492.713,A 0.000,B 0.000,C 90.000,E1 128.338} C_DIS
LIN {X -0.134,Y -296.141,Z 492.712,A 0.000,B 0.000,C 90.000,E1 128.177} C_DIS
LIN {X -0.003,Y -298.409,Z 492.711,A 0.000,B 0.000,C 90.000,E1 127.971} C_DIS
LIN {X -0.126,Y -302.282,Z 492.708,A 0.000,B 0.000,C 90.000,E1 127.523} C_DIS
LIN {X 0.080,Y -304.153,Z 492.707,A 0.000,B 0.000,C 90.000,E1 127.156} C_DIS
LIN {X -0.140,Y -305.617,Z 492.705,A 0.000,B 0.000,C 90.000,E1 126.870} C_DIS
LIN {X 0.087,Y -307.732,Z 492.701,A 0.000,B 0.000,C 90.000,E1 126.171} C_DIS
LIN {X -0.114,Y -317.903,Z 492.683,A 0.000,B 0.000,C 90.000,E1 122.959} C_DIS
LIN {X -0.061,Y -328.390,Z 492.667,A 0.000,B 0.000,C 90.000,E1 120.079} C_DIS
LIN {X -0.036,Y -340.243,Z 492.651,A 0.000,B 0.000,C 90.000,E1 117.257} C_DIS
LIN {X -0.144,Y -353.565,Z 492.636,A 0.000,B 0.000,C 90.000,E1 114.515} C_DIS
LIN {X 0.084,Y -366.741,Z 492.623,A 0.000,B 0.000,C 90.000,E1 112.078} C_DIS
LIN {X -0.106,Y -381.272,Z 492.610,A 0.000,B 0.000,C 90.000,E1 109.758} C_DIS
LIN {X -0.060,Y -397.262,Z 492.597,A 0.000,B 0.000,C 90.000,E1 107.457} C_DIS
LIN {X 0.153,Y -414.830,Z 492.585,A 0.000,B 0.000,C 90.000,E1 105.190} C_DIS
LIN {X -0.198,Y -434.072,Z 492.572,A 0.000,B 0.000,C 90.000,E1 103.063} C_DIS
LIN {X 0.019,Y -454.273,Z 492.561,A 0.000,B 0.000,C 90.000,E1 101.007} C_DIS
LIN {X -0.015,Y -475.013,Z 492.551,A 0.000,B 0.000,C 90.000,E1 99.151} C_DIS
LIN {X 0.163,Y -480.241,Z 492.548,A 0.000,B 0.000,C 90.000,E1 98.690} C_DIS
LIN {X -0.167,Y -482.325,Z 492.547,A 0.000,B 0.000,C 90.000,E1 98.511} C_DIS
LIN {X 0.188,Y -484.123,Z 492.546,A 0.000,B 0.000,C 90.000,E1 98.219} C_DIS
LIN {X -0.004,Y -485.473,Z 492.544,A 0.000,B 0.000,C 90.000,E1 97.992} C_DIS
LIN {X 0.185,Y -487.162,Z 492.542,A 0.000,B 0.000,C 90.000,E1 97.473} C_DIS
LIN {X -0.042,Y -487.771,Z 492.539,A 0.000,B 0.000,C 90.000,E1 97.004} C_DIS
LIN {X 0.163,Y -487.400,Z 492.536,A 0.000,B 0.000,C 90.000,E1 96.486} C_DIS
LIN {X -0.114,Y -485.989,Z 492.533,A 0.000,B 0.000,C 90.000,E1 96.024} C_DIS
LIN {X 0.206,Y -484.821,Z 492.532,A 0.000,B 0.000,C 90.000,E1 95.739} C_DIS
LIN {X 0.043,Y -483.258,Z 492.531,A 0.000,B 0.000,C 90.000,E1 95.511} C_DIS
LIN {X 0.213,Y -473.125,Z 492.524,A 0.000,B 0.000,C 90.000,E1 94.245} C_DIS
LIN {X -0.183,Y -459.456,Z 492.514,A 0.000,B 0.000,C 90.000,E1 92.522} C_DIS
LIN {X 0.047,Y -447.213,Z 492.504,A 0.000,B 0.000,C 90.000,E1 90.688} C_DIS
LIN {X 0.186,Y -434.112,Z 492.492,A 0.000,B 0.000,C 90.000,E1 88.568} C_DIS
LIN {X -0.126,Y -417.891,Z 492.477,A 0.000,B 0.000,C 90.000,E1 85.927} C_DIS
LIN {X -0.079,Y -403.574,Z 492.464,A 0.000,B 0.000,C 90.000,E1 83.451} C_DIS
LIN {X -0.054,Y -392.601,Z 492.453,A 0.000,B 0.000,C 90.000,E1 81.489} C_DIS
LIN {X -0.179,Y -383.185,Z 492.443,A 0.000,B 0.000,C 90.000,E1 79.803} C_DIS
LIN {X -0.011,Y -369.150,Z 492.429,A 0.000,B 0.000,C 90.000,E1 77.173} C_DIS
LIN {X 0.015,Y -358.840,Z 492.417,A 0.000,B 0.000,C 90.000,E1 75.102} C_DIS
LIN {X -0.144,Y -348.291,Z 492.404,A 0.000,B 0.000,C 90.000,E1 72.725} C_DIS
LIN {X -0.037,Y -335.641,Z 492.385,A 0.000,B 0.000,C 90.000,E1 69.337} C_DIS
LIN {X -0.115,Y -325.129,Z 492.368,A 0.000,B 0.000,C 90.000,E1 66.230} C_DIS
LIN {X -0.103,Y -316.989,Z 492.354,A 0.000,B 0.000,C 90.000,E1 63.691} C_DIS
LIN {X -0.007,Y -308.962,Z 492.339,A 0.000,B 0.000,C 90.000,E1 61.101} C_DIS
LIN {X 0.022,Y -300.990,Z 492.325,A 0.000,B 0.000,C 90.000,E1 58.486} C_DIS
LIN {X -0.029,Y -291.421,Z 492.307,A 0.000,B 0.000,C 90.000,E1 55.182} C_DIS
LIN {X 0.030,Y -284.159,Z 492.292,A 0.000,B 0.000,C 90.000,E1 52.477} C_DIS
LIN {X 0.013,Y -278.651,Z 492.280,A 0.000,B 0.000,C 90.000,E1 50.436} C_DIS
LIN {X -0.143,Y -272.723,Z 492.269,A 0.000,B 0.000,C 90.000,E1 48.405} C_DIS
LIN {X -0.005,Y -268.495,Z 492.261,A 0.000,B 0.000,C 90.000,E1 46.986} C_DIS
LIN {X -0.053,Y -262.938,Z 492.251,A 0.000,B 0.000,C 90.000,E1 45.243} C_DIS
LIN {X -0.130,Y -254.923,Z 492.237,A 0.000,B 0.000,C 90.000,E1 42.771} C_DIS
LIN {X -0.002,Y -246.067,Z 492.221,A 0.000,B 0.000,C 90.000,E1 39.850} C_DIS
LIN {X -0.012,Y -235.524,Z 492.201,A 0.000,B 0.000,C 90.000,E1 36.171} C_DIS
LIN {X 0.001,Y -227.794,Z 492.184,A 0.000,B 0.000,C 90.000,E1 33.166} C_DIS
LIN {X -0.045,Y -221.088,Z 492.167,A 0.000,B 0.000,C 90.000,E1 30.129} C_DIS
LIN {X 0.093,Y -215.160,Z 492.150,A 0.000,B 0.000,C 90.000,E1 27.001} C_DIS
LIN {X -0.011,Y -210.095,Z 492.133,A 0.000,B 0.000,C 90.000,E1 23.898} C_DIS
LIN {X -0.009,Y -204.851,Z 492.111,A 0.000,B 0.000,C 90.000,E1 19.939} C_DIS
LIN {X -0.068,Y -200.485,Z 492.089,A 0.000,B 0.000,C 90.000,E1 15.953} C_DIS
LIN {X 0.030,Y -196.643,Z 492.062,A 0.000,B 0.000,C 90.000,E1 11.074} C_DIS
LIN {X 0.097,Y -193.744,Z 492.025,A 0.000,B 0.000,C 90.000,E1 4.531} C_DIS
LIN {X -0.093,Y -195.068,Z 491.956,A 0.000,B 0.000,C 90.000,E1 352.186} C_DIS
LIN {X -0.059,Y -198.197,Z 491.929,A 0.000,B 0.000,C 90.000,E1 347.285} C_DIS
LIN {X -0.007,Y -202.740,Z 491.902,A 0.000,B 0.000,C 90.000,E1 342.417} C_DIS
LIN {X -0.006,Y -207.507,Z 491.880,A 0.000,B 0.000,C 90.000,E1 338.411} C_DIS
LIN {X -0.049,Y -213.023,Z 491.858,A 0.000,B 0.000,C 90.000,E1 334.460} C_DIS
LIN {X -0.027,Y -219.182,Z 491.836,A 0.000,B 0.000,C 90.000,E1 330.539} C_DIS
LIN {X -0.150,Y -225.919,Z 491.815,A 0.000,B 0.000,C 90.000,E1 326.707} C_DIS
LIN {X 0.071,Y -233.298,Z 491.794,A 0.000,B 0.000,C 90.000,E1 322.844} C_DIS
LIN {X 0.073,Y -241.487,Z 491.773,A 0.000,B 0.000,C 90.000,E1 319.094} C_DIS
LIN {X 0.089,Y -250.737,Z 491.752,A 0.000,B 0.000,C 90.000,E1 315.405} C_DIS
LIN {X -0.106,Y -261.396,Z 491.732,A 0.000,B 0.000,C 90.000,E1 311.838} C_DIS
LIN {X 0.038,Y -271.843,Z 491.715,A 0.000,B 0.000,C 90.000,E1 308.624} C_DIS
LIN {X -0.067,Y -284.733,Z 491.695,A 0.000,B 0.000,C 90.000,E1 305.185} C_DIS
LIN {X -0.026,Y -297.269,Z 491.678,A 0.000,B 0.000,C 90.000,E1 302.133} C_DIS
LIN {X 0.003,Y -310.565,Z 491.662,A 0.000,B 0.000,C 90.000,E1 299.155} C_DIS
LIN {X 0.038,Y -320.148,Z 491.651,A 0.000,B 0.000,C 90.000,E1 297.206} C_DIS
LIN {X 0.178,Y -334.155,Z 491.637,A 0.000,B 0.000,C 90.000,E1 294.643} C_DIS
LIN {X -0.056,Y -349.728,Z 491.623,A 0.000,B 0.000,C 90.000,E1 292.206} C_DIS
LIN {X -0.106,Y -369.160,Z 491.608,A 0.000,B 0.000,C 90.000,E1 289.504} C_DIS
LIN {X 0.017,Y -388.173,Z 491.595,A 0.000,B 0.000,C 90.000,E1 287.149} C_DIS
LIN {X 0.008,Y -413.051,Z 491.580,A 0.000,B 0.000,C 90.000,E1 284.356} C_DIS
LIN {X -0.063,Y -428.096,Z 491.571,A 0.000,B 0.000,C 90.000,E1 282.771} C_DIS
LIN {X 0.105,Y -440.418,Z 491.564,A 0.000,B 0.000,C 90.000,E1 281.422} C_DIS
LIN {X 0.108,Y -449.941,Z 491.558,A 0.000,B 0.000,C 90.000,E1 280.366} C_DIS
LIN {X -0.127,Y -456.528,Z 491.553,A 0.000,B 0.000,C 90.000,E1 279.613} C_DIS
LIN {X 0.158,Y -462.475,Z 491.549,A 0.000,B 0.000,C 90.000,E1 278.803} C_DIS
LIN {X 0.037,Y -467.913,Z 491.545,A 0.000,B 0.000,C 90.000,E1 278.049} C_DIS
LIN {X -0.036,Y -472.797,Z 491.540,A 0.000,B 0.000,C 90.000,E1 277.296} C_DIS
LIN {X 0.203,Y -478.410,Z 491.535,A 0.000,B 0.000,C 90.000,E1 276.258} C_DIS
LIN {X 0.165,Y -481.951,Z 491.531,A 0.000,B 0.000,C 90.000,E1 275.511} C_DIS
LIN {X -0.147,Y -483.986,Z 491.528,A 0.000,B 0.000,C 90.000,E1 275.049} C_DIS
LIN {X 0.026,Y -485.709,Z 491.525,A 0.000,B 0.000,C 90.000,E1 274.531} C_DIS
LIN {X 0.210,Y -487.161,Z 491.522,A 0.000,B 0.000,C 90.000,E1 274.012} C_DIS
LIN {X -0.117,Y -488.266,Z 491.520,A 0.000,B 0.000,C 90.000,E1 273.555} C_DIS
LIN {X 0.083,Y -489.070,Z 491.517,A 0.000,B 0.000,C 90.000,E1 273.037} C_DIS
LIN {X -0.226,Y -489.502,Z 491.514,A 0.000,B 0.000,C 90.000,E1 272.579} C_DIS
LIN {X -0.038,Y -489.579,Z 491.511,A 0.000,B 0.000,C 90.000,E1 272.064} C_DIS
LIN {X 0.168,Y -489.262,Z 491.509,A 0.000,B 0.000,C 90.000,E1 271.547} C_DIS
LIN {X -0.130,Y -488.498,Z 491.506,A 0.000,B 0.000,C 90.000,E1 271.088} C_DIS
LIN {X 0.060,Y -487.234,Z 491.503,A 0.000,B 0.000,C 90.000,E1 270.573} C_DIS
LIN {X -0.240,Y -485.378,Z 491.500,A 0.000,B 0.000,C 90.000,E1 270.115} C_DIS
LIN {X -0.061,Y -482.863,Z 491.498,A 0.000,B 0.000,C 90.000,E1 269.599} C_DIS
LIN {X -0.221,Y -481.393,Z 491.496,A 0.000,B 0.000,C 90.000,E1 269.370} C_DIS
LIN {X -0.069,Y -477.672,Z 491.494,A 0.000,B 0.000,C 90.000,E1 268.854} C_DIS
LIN {X 0.059,Y -473.076,Z 491.491,A 0.000,B 0.000,C 90.000,E1 268.339} C_DIS
LIN {X -0.102,Y -470.386,Z 491.489,A 0.000,B 0.000,C 90.000,E1 268.108} C_DIS
LIN {X -0.219,Y -464.319,Z 491.487,A 0.000,B 0.000,C 90.000,E1 267.650} C_DIS
LIN {X 0.196,Y -457.791,Z 491.485,A 0.000,B 0.000,C 90.000,E1 267.192} C_DIS
LIN {X 0.208,Y -454.651,Z 491.484,A 0.000,B 0.000,C 90.000,E1 267.020} C_DIS
LIN {X 0.050,Y -447.832,Z 491.482,A 0.000,B 0.000,C 90.000,E1 266.731} C_DIS
LIN {X -0.156,Y -440.921,Z 491.480,A 0.000,B 0.000,C 90.000,E1 266.502} C_DIS
LIN {X -0.029,Y -433.497,Z 491.479,A 0.000,B 0.000,C 90.000,E1 266.274} C_DIS
LIN {X 0.019,Y -425.006,Z 491.478,A 0.000,B 0.000,C 90.000,E1 266.102} C_DIS
LIN {X 0.013,Y -414.411,Z 491.478,A 0.000,B 0.000,C 90.000,E1 265.988} C_DIS
LIN {X -0.150,Y -409.862,Z 491.478,A 0.000,B 0.000,C 90.000,E1 265.988} C_DIS
LIN {X 0.078,Y -180.919,Z 491.478,A 0.000,B 0.000,C 90.000,E1 265.931} C_DIS
LIN {X -0.063,Y -180.845,Z 491.472,A 0.000,B 0.000,C 90.000,E1 264.951} C_DIS
LIN {X 0.015,Y -178.889,Z 491.443,A 0.000,B 0.000,C 90.000,E1 259.690} C_DIS
LIN {X 0.090,Y -175.932,Z 491.414,A 0.000,B 0.000,C 90.000,E1 254.574} C_DIS
LIN {X 0.035,Y -175.377,Z 491.410,A 0.000,B 0.000,C 90.000,E1 253.740} C_DIS
LIN {X 0.032,Y -172.152,Z 491.386,A 0.000,B 0.000,C 90.000,E1 249.464} C_DIS
LIN {X 0.070,Y -171.618,Z 491.381,A 0.000,B 0.000,C 90.000,E1 248.592} C_DIS
LIN {X 0.058,Y -167.841,Z 491.357,A 0.000,B 0.000,C 90.000,E1 244.280} C_DIS
LIN {X -0.002,Y -166.568,Z 491.348,A 0.000,B 0.000,C 90.000,E1 242.564} C_DIS
LIN {X -0.015,Y -162.562,Z 491.323,A 0.000,B 0.000,C 90.000,E1 238.201} C_DIS
LIN {X 0.044,Y -161.241,Z 491.314,A 0.000,B 0.000,C 90.000,E1 236.421} C_DIS
LIN {X -0.045,Y -157.245,Z 491.289,A 0.000,B 0.000,C 90.000,E1 232.029} C_DIS
LIN {X 0.001,Y -155.969,Z 491.279,A 0.000,B 0.000,C 90.000,E1 230.231} C_DIS
LIN {X 0.059,Y -152.223,Z 491.254,A 0.000,B 0.000,C 90.000,E1 225.729} C_DIS
LIN {X -0.030,Y -150.467,Z 491.239,A 0.000,B 0.000,C 90.000,E1 223.056} C_DIS
LIN {X -0.010,Y -147.192,Z 491.214,A 0.000,B 0.000,C 90.000,E1 218.508} C_DIS
LIN {X 0.071,Y -145.210,Z 491.194,A 0.000,B 0.000,C 90.000,E1 214.818} C_DIS
LIN {X -0.019,Y -142.344,Z 491.163,A 0.000,B 0.000,C 90.000,E1 209.333} C_DIS
LIN {X 0.034,Y -141.732,Z 491.153,A 0.000,B 0.000,C 90.000,E1 207.462} C_DIS
LIN {X 0.016,Y -139.483,Z 491.117,A 0.000,B 0.000,C 90.000,E1 200.972} C_DIS
LIN {X 0.005,Y -138.982,Z 491.101,A 0.000,B 0.000,C 90.000,E1 198.181} C_DIS
LIN {X -0.034,Y -138.334,Z 491.054,A 0.000,B 0.000,C 90.000,E1 189.792} C_DIS
LIN {X -0.009,Y -139.426,Z 491.008,A 0.000,B 0.000,C 90.000,E1 181.375} C_DIS
LIN {X 0.044,Y -141.351,Z 490.971,A 0.000,B 0.000,C 90.000,E1 174.837} C_DIS
LIN {X 0.021,Y -142.705,Z 490.956,A 0.000,B 0.000,C 90.000,E1 172.064} C_DIS
LIN {X -0.020,Y -145.076,Z 490.930,A 0.000,B 0.000,C 90.000,E1 167.465} C_DIS
LIN {X -0.024,Y -147.701,Z 490.910,A 0.000,B 0.000,C 90.000,E1 163.795} C_DIS
LIN {X 0.009,Y -150.353,Z 490.890,A 0.000,B 0.000,C 90.000,E1 160.134} C_DIS
LIN {X 0.002,Y -154.608,Z 490.865,A 0.000,B 0.000,C 90.000,E1 155.613} C_DIS
LIN {X 0.008,Y -158.150,Z 490.845,A 0.000,B 0.000,C 90.000,E1 152.025} C_DIS
LIN {X 0.053,Y -162.436,Z 490.825,A 0.000,B 0.000,C 90.000,E1 148.456} C_DIS
LIN {X -0.051,Y -166.696,Z 490.805,A 0.000,B 0.000,C 90.000,E1 144.975} C_DIS
LIN {X 0.061,Y -171.702,Z 490.786,A 0.000,B 0.000,C 90.000,E1 141.457} C_DIS
LIN {X -0.004,Y -176.675,Z 490.767,A 0.000,B 0.000,C 90.000,E1 138.038} C_DIS
LIN {X -0.009,Y -180.971,Z 490.753,A 0.000,B 0.000,C 90.000,E1 135.486} C_DIS
LIN {X -0.022,Y -186.396,Z 490.734,A 0.000,B 0.000,C 90.000,E1 132.123} C_DIS
LIN {X -0.083,Y -191.024,Z 490.720,A 0.000,B 0.000,C 90.000,E1 129.644} C_DIS
LIN {X 0.071,Y -193.182,Z 490.713,A 0.000,B 0.000,C 90.000,E1 128.302} C_DIS
LIN {X 0.076,Y -290.611,Z 490.713,A 0.000,B 0.000,C 90.000,E1 128.302} C_DIS
LIN {X -0.106,Y -292.520,Z 490.713,A 0.000,B 0.000,C 90.000,E1 128.302} C_DIS
LIN {X -0.008,Y -298.035,Z 490.711,A 0.000,B 0.000,C 90.000,E1 127.971} C_DIS
LIN {X 0.092,Y -301.227,Z 490.709,A 0.000,B 0.000,C 90.000,E1 127.604} C_DIS
LIN {X 0.008,Y -303.224,Z 490.707,A 0.000,B 0.000,C 90.000,E1 127.317} C_DIS
LIN {X -0.079,Y -304.795,Z 490.706,A 0.000,B 0.000,C 90.000,E1 127.030} C_DIS
LIN {X 0.123,Y -306.151,Z 490.704,A 0.000,B 0.000,C 90.000,E1 126.664} C_DIS
LIN {X -0.077,Y -312.081,Z 490.693,A 0.000,B 0.000,C 90.000,E1 124.739} C_DIS
LIN {X -0.056,Y -322.936,Z 490.675,A 0.000,B 0.000,C 90.000,E1 121.514} C_DIS
LIN {X -0.198,Y -334.091,Z 490.659,A 0.000,B 0.000,C 90.000,E1 118.693} C_DIS
LIN {X 0.136,Y -346.659,Z 490.644,A 0.000,B 0.000,C 90.000,E1 115.848} C_DIS
LIN {X -0.131,Y -359.114,Z 490.630,A 0.000,B 0.000,C 90.000,E1 113.462} C_DIS
LIN {X 0.109,Y -372.867,Z 490.617,A 0.000,B 0.000,C 90.000,E1 111.046} C_DIS
LIN {X 0.081,Y -388.017,Z 490.604,A 0.000,B 0.000,C 90.000,E1 108.725} C_DIS
LIN {X 0.183,Y -404.679,Z 490.591,A 0.000,B 0.000,C 90.000,E1 106.441} C_DIS
LIN {X 0.083,Y -422.972,Z 490.579,A 0.000,B 0.000,C 90.000,E1 104.245} C_DIS
LIN {X 0.111,Y -442.759,Z 490.567,A 0.000,B 0.000,C 90.000,E1 102.119} C_DIS
LIN {X -0.136,Y -463.205,Z 490.557,A 0.000,B 0.000,C 90.000,E1 100.197} C_DIS
LIN {X -0.176,Y -481.333,Z 490.548,A 0.000,B 0.000,C 90.000,E1 98.624} C_DIS
LIN {X -0.192,Y -483.271,Z 490.547,A 0.000,B 0.000,C 90.000,E1 98.398} C_DIS
LIN {X -0.136,Y -484.755,Z 490.545,A 0.000,B 0.000,C 90.000,E1 98.163} C_DIS
LIN {X 0.227,Y -485.980,Z 490.544,A 0.000,B 0.000,C 90.000,E1 97.871} C_DIS
LIN {X 0.044,Y -486.876,Z 490.542,A 0.000,B 0.000,C 90.000,E1 97.644} C_DIS
LIN {X -0.240,Y -487.834,Z 490.540,A 0.000,B 0.000,C 90.000,E1 97.182} C_DIS
LIN {X -0.035,Y -487.799,Z 490.537,A 0.000,B 0.000,C 90.000,E1 96.663} C_DIS
LIN {X 0.176,Y -486.762,Z 490.534,A 0.000,B 0.000,C 90.000,E1 96.144} C_DIS
LIN {X 0.064,Y -485.821,Z 490.533,A 0.000,B 0.000,C 90.000,E1 95.910} C_DIS
LIN {X -0.098,Y -484.539,Z 490.531,A 0.000,B 0.000,C 90.000,E1 95.682} C_DIS
LIN {X -0.216,Y -482.824,Z 490.530,A 0.000,B 0.000,C 90.000,E1 95.448} C_DIS
LIN {X 0.112,Y -464.721,Z 490.518,A 0.000,B 0.000,C 90.000,E1 93.154} C_DIS
LIN {X -0.215,Y -453.635,Z 490.509,A 0.000,B 0.000,C 90.000,E1 91.661} C_DIS
LIN {X -0.009,Y -436.983,Z 490.495,A 0.000,B 0.000,C 90.000,E1 89.026} C_DIS
LIN {X -0.099,Y -423.910,Z 490.483,A 0.000,B 0.000,C 90.000,E1 86.906} C_DIS
LIN {X -0.110,Y -412.680,Z 490.472,A 0.000,B 0.000,C 90.000,E1 85.008} C_DIS
LIN {X 0.149,Y -400.045,Z 490.460,A 0.000,B 0.000,C 90.000,E1 82.761} C_DIS
LIN {X 0.089,Y -390.647,Z 490.451,A 0.000,B 0.000,C 90.000,E1 81.084} C_DIS
LIN {X -0.073,Y -381.230,Z 490.441,A 0.000,B 0.000,C 90.000,E1 79.398} C_DIS
LIN {X 0.115,Y -367.291,Z 490.427,A 0.000,B 0.000,C 90.000,E1 76.756} C_DIS
LIN {X 0.009,Y -357.147,Z 490.415,A 0.000,B 0.000,C 90.000,E1 74.700} C_DIS
LIN {X -0.099,Y -346.780,Z 490.402,A 0.000,B 0.000,C 90.000,E1 72.308} C_DIS
LIN {X 0.070,Y -334.284,Z 490.383,A 0.000,B 0.000,C 90.000,E1 68.901} C_DIS
LIN {X -0.050,Y -323.798,Z 490.365,A 0.000,B 0.000,C 90.000,E1 65.793} C_DIS
LIN {X -0.076,Y -315.644,Z 490.351,A 0.000,B 0.000,C 90.000,E1 63.256} C_DIS
LIN {X -0.023,Y -307.591,Z 490.337,A 0.000,B 0.000,C 90.000,E1 60.667} C_DIS
LIN {X 0.020,Y -299.624,Z 490.322,A 0.000,B 0.000,C 90.000,E1 58.043} C_DIS
LIN {X 0.180,Y -290.104,Z 490.304,A 0.000,B 0.000,C 90.000,E1 54.689} C_DIS
LIN {X -0.023,Y -282.845,Z 490.289,A 0.000,B 0.000,C 90.000,E1 52.029} C_DIS
LIN {X -0.063,Y -277.220,Z 490.278,A 0.000,B 0.000,C 90.000,E1 49.989} C_DIS
LIN {X -0.052,Y -273.283,Z 490.270,A 0.000,B 0.000,C 90.000,E1 48.609} C_DIS
LIN {X -0.125,Y -266.908,Z 490.258,A 0.000,B 0.000,C 90.000,E1 46.539} C_DIS
LIN {X -0.151,Y -260.177,Z 490.247,A 0.000,B 0.000,C 90.000,E1 44.433} C_DIS
LIN {X 0.107,Y -250.002,Z 490.229,A 0.000,B 0.000,C 90.000,E1 41.148} C_DIS
LIN {X -0.020,Y -240.281,Z 490.210,A 0.000,B 0.000,C 90.000,E1 37.890} C_DIS
LIN {X 0.057,Y -232.139,Z 490.194,A 0.000,B 0.000,C 90.000,E1 34.898} C_DIS
LIN {X 0.048,Y -224.822,Z 490.177,A 0.000,B 0.000,C 90.000,E1 31.878} C_DIS
LIN {X 0.005,Y -218.471,Z 490.160,A 0.000,B 0.000,C 90.000,E1 28.821} C_DIS
LIN {X -0.021,Y -212.904,Z 490.143,A 0.000,B 0.000,C 90.000,E1 25.720} C_DIS
LIN {X -0.073,Y -208.194,Z 490.125,A 0.000,B 0.000,C 90.000,E1 22.589} C_DIS
LIN {X -0.013,Y -203.258,Z 490.103,A 0.000,B 0.000,C 90.000,E1 18.598} C_DIS
LIN {X -0.049,Y -199.198,Z 490.081,A 0.000,B 0.000,C 90.000,E1 14.592} C_DIS
LIN {X -0.040,Y -195.785,Z 490.054,A 0.000,B 0.000,C 90.000,E1 9.726} C_DIS
LIN {X 0.037,Y -193.203,Z 490.013,A 0.000,B 0.000,C 90.000,E1 2.350} C_DIS
LIN {X -0.047,Y -194.561,Z 489.961,A 0.000,B 0.000,C 90.000,E1 352.989} C_DIS
LIN {X 0.099,Y -197.439,Z 489.934,A 0.000,B 0.000,C 90.000,E1 348.049} C_DIS
LIN {X 0.071,Y -201.746,Z 489.907,A 0.000,B 0.000,C 90.000,E1 343.196} C_DIS
LIN {X -0.026,Y -206.355,Z 489.884,A 0.000,B 0.000,C 90.000,E1 339.209} C_DIS
LIN {X 0.002,Y -211.713,Z 489.862,A 0.000,B 0.000,C 90.000,E1 335.229} C_DIS
LIN {X -0.014,Y -217.783,Z 489.841,A 0.000,B 0.000,C 90.000,E1 331.307} C_DIS
LIN {X -0.099,Y -224.366,Z 489.819,A 0.000,B 0.000,C 90.000,E1 327.454} C_DIS
LIN {X -0.060,Y -231.621,Z 489.798,A 0.000,B 0.000,C 90.000,E1 323.623} C_DIS
LIN {X 0.076,Y -239.639,Z 489.777,A 0.000,B 0.000,C 90.000,E1 319.828} C_DIS
LIN {X 0.049,Y -248.694,Z 489.756,A 0.000,B 0.000,C 90.000,E1 316.134} C_DIS
LIN {X 0.116,Y -258.027,Z 489.738,A 0.000,B 0.000,C 90.000,E1 312.852} C_DIS
LIN {X -0.002,Y -269.388,Z 489.718,A 0.000,B 0.000,C 90.000,E1 309.322} C_DIS
LIN {X -0.034,Y -282.075,Z 489.699,A 0.000,B 0.000,C 90.000,E1 305.851} C_DIS
LIN {X -0.087,Y -295.852,Z 489.680,A 0.000,B 0.000,C 90.000,E1 302.467} C_DIS
LIN {X 0.043,Y -309.057,Z 489.664,A 0.000,B 0.000,C 90.000,E1 299.461} C_DIS
LIN {X 0.043,Y -318.497,Z 489.653,A 0.000,B 0.000,C 90.000,E1 297.513} C_DIS
LIN {X -0.005,Y -332.362,Z 489.639,A 0.000,B 0.000,C 90.000,E1 294.975} C_DIS
LIN {X -0.150,Y -347.717,Z 489.625,A 0.000,B 0.000,C 90.000,E1 292.514} C_DIS
LIN {X 0.088,Y -366.929,Z 489.610,A 0.000,B 0.000,C 90.000,E1 289.758} C_DIS
LIN {X 0.173,Y -385.783,Z 489.597,A 0.000,B 0.000,C 90.000,E1 287.402} C_DIS
LIN {X 0.043,Y -410.764,Z 489.581,A 0.000,B 0.000,C 90.000,E1 284.592} C_DIS
LIN {X -0.211,Y -426.041,Z 489.572,A 0.000,B 0.000,C 90.000,E1 283.008} C_DIS
LIN {X 0.176,Y -438.179,Z 489.565,A 0.000,B 0.000,C 90.000,E1 281.658} C_DIS
LIN {X 0.174,Y -447.838,Z 489.559,A 0.000,B 0.000,C 90.000,E1 280.602} C_DIS
LIN {X -0.069,Y -454.572,Z 489.555,A 0.000,B 0.000,C 90.000,E1 279.849} C_DIS
LIN {X -0.189,Y -460.769,Z 489.550,A 0.000,B 0.000,C 90.000,E1 279.086} C_DIS
LIN {X -0.104,Y -468.112,Z 489.545,A 0.000,B 0.000,C 90.000,E1 278.049} C_DIS
LIN {X -0.176,Y -472.971,Z 489.540,A 0.000,B 0.000,C 90.000,E1 277.296} C_DIS
LIN {X 0.259,Y -477.284,Z 489.536,A 0.000,B 0.000,C 90.000,E1 276.486} C_DIS
LIN {X 0.211,Y -481.025,Z 489.532,A 0.000,B 0.000,C 90.000,E1 275.739} C_DIS
LIN {X 0.196,Y -484.171,Z 489.528,A 0.000,B 0.000,C 90.000,E1 274.992} C_DIS
LIN {X -0.111,Y -485.920,Z 489.525,A 0.000,B 0.000,C 90.000,E1 274.531} C_DIS
LIN {X 0.073,Y -487.336,Z 489.522,A 0.000,B 0.000,C 90.000,E1 274.012} C_DIS
LIN {X 0.235,Y -488.443,Z 489.520,A 0.000,B 0.000,C 90.000,E1 273.498} C_DIS
LIN {X -0.052,Y -489.246,Z 489.517,A 0.000,B 0.000,C 90.000,E1 273.037} C_DIS
LIN {X 0.128,Y -489.681,Z 489.514,A 0.000,B 0.000,C 90.000,E1 272.522} C_DIS
LIN {X -0.171,Y -489.746,Z 489.511,A 0.000,B 0.000,C 90.000,E1 272.064} C_DIS
LIN {X 0.035,Y -489.421,Z 489.509,A 0.000,B 0.000,C 90.000,E1 271.547} C_DIS
LIN {X 0.228,Y -488.652,Z 489.506,A 0.000,B 0.000,C 90.000,E1 271.031} C_DIS
LIN {X -0.069,Y -487.345,Z 489.503,A 0.000,B 0.000,C 90.000,E1 270.573} C_DIS
LIN {X 0.117,Y -485.506,Z 489.500,A 0.000,B 0.000,C 90.000,E1 270.057} C_DIS
LIN {X -0.036,Y -484.327,Z 489.499,A 0.000,B 0.000,C 90.000,E1 269.828} C_DIS
LIN {X 0.134,Y -481.426,Z 489.496,A 0.000,B 0.000,C 90.000,E1 269.312} C_DIS
LIN {X -0.027,Y -479.707,Z 489.495,A 0.000,B 0.000,C 90.000,E1 269.083} C_DIS
LIN {X 0.114,Y -475.548,Z 489.492,A 0.000,B 0.000,C 90.000,E1 268.568} C_DIS
LIN {X -0.225,Y -470.289,Z 489.489,A 0.000,B 0.000,C 90.000,E1 268.108} C_DIS
LIN {X 0.199,Y -464.412,Z 489.487,A 0.000,B 0.000,C 90.000,E1 267.593} C_DIS
LIN {X 0.137,Y -457.833,Z 489.484,A 0.000,B 0.000,C 90.000,E1 267.192} C_DIS
LIN {X 0.150,Y -450.933,Z 489.483,A 0.000,B 0.000,C 90.000,E1 266.849} C_DIS
LIN {X -0.215,Y -444.142,Z 489.481,A 0.000,B 0.000,C 90.000,E1 266.617} C_DIS
LIN {X 0.171,Y -436.885,Z 489.480,A 0.000,B 0.000,C 90.000,E1 266.331} C_DIS
LIN {X 0.018,Y -428.511,Z 489.479,A 0.000,B 0.000,C 90.000,E1 266.159} C_DIS
LIN {X -0.103,Y -419.475,Z 489.478,A 0.000,B 0.000,C 90.000,E1 266.045} C_DIS
LIN {X -0.168,Y -409.957,Z 489.478,A 0.000,B 0.000,C 90.000,E1 265.988} C_DIS
LIN {X 0.071,Y -180.918,Z 489.478,A 0.000,B 0.000,C 90.000,E1 265.931} C_DIS
LIN {X -0.069,Y -180.844,Z 489.472,A 0.000,B 0.000,C 90.000,E1 264.951} C_DIS
LIN {X 0.007,Y -178.888,Z 489.443,A 0.000,B 0.000,C 90.000,E1 259.690} C_DIS
LIN {X 0.083,Y -175.931,Z 489.414,A 0.000,B 0.000,C 90.000,E1 254.574} C_DIS
LIN {X 0.028,Y -175.376,Z 489.410,A 0.000,B 0.000,C 90.000,E1 253.740} C_DIS
LIN {X 0.026,Y -172.151,Z 489.386,A 0.000,B 0.000,C 90.000,E1 249.464} C_DIS
LIN {X 0.064,Y -171.616,Z 489.381,A 0.000,B 0.000,C 90.000,E1 248.592} C_DIS
LIN {X 0.052,Y -167.840,Z 489.357,A 0.000,B 0.000,C 90.000,E1 244.280} C_DIS
LIN {X -0.008,Y -166.567,Z 489.348,A 0.000,B 0.000,C 90.000,E1 242.564} C_DIS
LIN {X -0.022,Y -162.560,Z 489.323,A 0.000,B 0.000,C 90.000,E1 238.201} C_DIS
LIN {X 0.038,Y -161.240,Z 489.314,A 0.000,B 0.000,C 90.000,E1 236.421} C_DIS
LIN {X 0.072,Y -157.244,Z 489.289,A 0.000,B 0.000,C 90.000,E1 231.984} C_DIS
LIN {X -0.004,Y -155.967,Z 489.279,A 0.000,B 0.000,C 90.000,E1 230.231} C_DIS
LIN {X 0.054,Y -152.222,Z 489.254,A 0.000,B 0.000,C 90.000,E1 225.729} C_DIS
LIN {X -0.036,Y -150.465,Z 489.239,A 0.000,B 0.000,C 90.000,E1 223.056} C_DIS
LIN {X -0.015,Y -147.190,Z 489.214,A 0.000,B 0.000,C 90.000,E1 218.508} C_DIS
LIN {X 0.066,Y -145.209,Z 489.194,A 0.000,B 0.000,C 90.000,E1 214.818} C_DIS
LIN {X -0.024,Y -142.343,Z 489.163,A 0.000,B 0.000,C 90.000,E1 209.333} C_DIS
LIN {X 0.029,Y -141.731,Z 489.153,A 0.000,B 0.000,C 90.000,E1 207.462} C_DIS
LIN {X 0.011,Y -139.483,Z 489.117,A 0.000,B 0.000,C 90.000,E1 200.972} C_DIS
LIN {X -0.001,Y -138.982,Z 489.101,A 0.000,B 0.000,C 90.000,E1 198.181} C_DIS
LIN {X -0.039,Y -138.333,Z 489.054,A 0.000,B 0.000,C 90.000,E1 189.792} C_DIS
LIN {X -0.015,Y -139.427,Z 489.008,A 0.000,B 0.000,C 90.000,E1 181.375} C_DIS
LIN {X 0.039,Y -141.351,Z 488.971,A 0.000,B 0.000,C 90.000,E1 174.837} C_DIS
LIN {X 0.015,Y -142.705,Z 488.956,A 0.000,B 0.000,C 90.000,E1 172.064} C_DIS
LIN {X -0.025,Y -145.078,Z 488.930,A 0.000,B 0.000,C 90.000,E1 167.465} C_DIS
LIN {X -0.030,Y -147.703,Z 488.910,A 0.000,B 0.000,C 90.000,E1 163.795} C_DIS
LIN {X 0.054,Y -150.356,Z 488.890,A 0.000,B 0.000,C 90.000,E1 160.115} C_DIS
LIN {X 0.073,Y -153.779,Z 488.870,A 0.000,B 0.000,C 90.000,E1 156.485} C_DIS
LIN {X -0.007,Y -157.191,Z 488.850,A 0.000,B 0.000,C 90.000,E1 152.922} C_DIS
LIN {X 0.075,Y -161.351,Z 488.830,A 0.000,B 0.000,C 90.000,E1 149.331} C_DIS
LIN {X 0.087,Y -165.554,Z 488.810,A 0.000,B 0.000,C 90.000,E1 145.801} C_DIS
LIN {X -0.029,Y -170.469,Z 488.791,A 0.000,B 0.000,C 90.000,E1 142.351} C_DIS
LIN {X -0.011,Y -175.350,Z 488.772,A 0.000,B 0.000,C 90.000,E1 138.895} C_DIS
LIN {X -0.016,Y -180.975,Z 488.753,A 0.000,B 0.000,C 90.000,E1 135.486} C_DIS
LIN {X -0.029,Y -186.399,Z 488.734,A 0.000,B 0.000,C 90.000,E1 132.123} C_DIS
LIN {X -0.089,Y -191.027,Z 488.720,A 0.000,B 0.000,C 90.000,E1 129.644} C_DIS
LIN {X 0.070,Y -193.260,Z 488.713,A 0.000,B 0.000,C 90.000,E1 128.257} C_DIS
LIN {X 0.053,Y -291.047,Z 488.713,A 0.000,B 0.000,C 90.000,E1 128.257} C_DIS
LIN {X -0.106,Y -292.591,Z 488.712,A 0.000,B 0.000,C 90.000,E1 128.257} C_DIS
LIN {X -0.018,Y -297.623,Z 488.711,A 0.000,B 0.000,C 90.000,E1 127.971} C_DIS
LIN {X -0.064,Y -300.862,Z 488.709,A 0.000,B 0.000,C 90.000,E1 127.649} C_DIS
LIN {X -0.081,Y -304.469,Z 488.706,A 0.000,B 0.000,C 90.000,E1 127.076} C_DIS
LIN {X -0.071,Y -305.923,Z 488.704,A 0.000,B 0.000,C 90.000,E1 126.744} C_DIS
LIN {X 0.124,Y -307.070,Z 488.702,A 0.000,B 0.000,C 90.000,E1 126.377} C_DIS
LIN {X -0.099,Y -317.155,Z 488.684,A 0.000,B 0.000,C 90.000,E1 123.166} C_DIS
LIN {X 0.099,Y -327.545,Z 488.668,A 0.000,B 0.000,C 90.000,E1 120.256} C_DIS
LIN {X -0.060,Y -339.297,Z 488.652,A 0.000,B 0.000,C 90.000,E1 117.462} C_DIS
LIN {X -0.041,Y -352.508,Z 488.637,A 0.000,B 0.000,C 90.000,E1 114.695} C_DIS
LIN {X 0.019,Y -365.579,Z 488.624,A 0.000,B 0.000,C 90.000,E1 112.280} C_DIS
LIN {X -0.061,Y -379.995,Z 488.611,A 0.000,B 0.000,C 90.000,E1 109.939} C_DIS
LIN {X -0.046,Y -395.862,Z 488.598,A 0.000,B 0.000,C 90.000,E1 107.638} C_DIS
LIN {X 0.133,Y -413.296,Z 488.586,A 0.000,B 0.000,C 90.000,E1 105.371} C_DIS
LIN {X -0.162,Y -432.407,Z 488.573,A 0.000,B 0.000,C 90.000,E1 103.231} C_DIS
LIN {X -0.158,Y -452.562,Z 488.562,A 0.000,B 0.000,C 90.000,E1 101.186} C_DIS
LIN {X 0.239,Y -473.262,Z 488.552,A 0.000,B 0.000,C 90.000,E1 99.265} C_DIS
LIN {X 0.053,Y -481.062,Z 488.548,A 0.000,B 0.000,C 90.000,E1 98.624} C_DIS
LIN {X 0.080,Y -483.069,Z 488.547,A 0.000,B 0.000,C 90.000,E1 98.398} C_DIS
LIN {X 0.179,Y -484.608,Z 488.545,A 0.000,B 0.000,C 90.000,E1 98.163} C_DIS
LIN {X -0.005,Y -485.914,Z 488.544,A 0.000,B 0.000,C 90.000,E1 97.936} C_DIS
LIN {X -0.123,Y -486.878,Z 488.543,A 0.000,B 0.000,C 90.000,E1 97.701} C_DIS
LIN {X 0.076,Y -487.951,Z 488.540,A 0.000,B 0.000,C 90.000,E1 97.182} C_DIS
LIN {X -0.203,Y -488.020,Z 488.537,A 0.000,B 0.000,C 90.000,E1 96.720} C_DIS
LIN {X 0.008,Y -487.096,Z 488.534,A 0.000,B 0.000,C 90.000,E1 96.201} C_DIS
LIN {X 0.218,Y -485.017,Z 488.532,A 0.000,B 0.000,C 90.000,E1 95.682} C_DIS
LIN {X 0.056,Y -483.407,Z 488.530,A 0.000,B 0.000,C 90.000,E1 95.454} C_DIS
LIN {X -0.105,Y -469.255,Z 488.521,A 0.000,B 0.000,C 90.000,E1 93.726} C_DIS
LIN {X -0.138,Y -455.948,Z 488.511,A 0.000,B 0.000,C 90.000,E1 91.949} C_DIS
LIN {X 0.217,Y -442.362,Z 488.499,A 0.000,B 0.000,C 90.000,E1 89.828} C_DIS
LIN {X 0.105,Y -430.895,Z 488.489,A 0.000,B 0.000,C 90.000,E1 87.993} C_DIS
LIN {X 0.002,Y -416.356,Z 488.475,A 0.000,B 0.000,C 90.000,E1 85.584} C_DIS
LIN {X -0.006,Y -402.061,Z 488.462,A 0.000,B 0.000,C 90.000,E1 83.109} C_DIS
LIN {X -0.028,Y -392.694,Z 488.452,A 0.000,B 0.000,C 90.000,E1 81.432} C_DIS
LIN {X -0.118,Y -381.711,Z 488.441,A 0.000,B 0.000,C 90.000,E1 79.454} C_DIS
LIN {X 0.075,Y -366.265,Z 488.425,A 0.000,B 0.000,C 90.000,E1 76.520} C_DIS
LIN {X 0.048,Y -356.212,Z 488.414,A 0.000,B 0.000,C 90.000,E1 74.448} C_DIS
LIN {X -0.097,Y -347.168,Z 488.402,A 0.000,B 0.000,C 90.000,E1 72.362} C_DIS
LIN {X 0.089,Y -334.583,Z 488.383,A 0.000,B 0.000,C 90.000,E1 68.954} C_DIS
LIN {X -0.015,Y -324.043,Z 488.366,A 0.000,B 0.000,C 90.000,E1 65.845} C_DIS
LIN {X -0.030,Y -315.858,Z 488.352,A 0.000,B 0.000,C 90.000,E1 63.307} C_DIS
LIN {X 0.034,Y -307.749,Z 488.337,A 0.000,B 0.000,C 90.000,E1 60.717} C_DIS
LIN {X -0.029,Y -297.794,Z 488.319,A 0.000,B 0.000,C 90.000,E1 57.454} C_DIS
LIN {X -0.005,Y -288.356,Z 488.301,A 0.000,B 0.000,C 90.000,E1 54.116} C_DIS
LIN {X -0.113,Y -282.903,Z 488.289,A 0.000,B 0.000,C 90.000,E1 52.110} C_DIS
LIN {X 0.027,Y -277.288,Z 488.278,A 0.000,B 0.000,C 90.000,E1 50.033} C_DIS
LIN {X 0.067,Y -273.343,Z 488.270,A 0.000,B 0.000,C 90.000,E1 48.647} C_DIS
LIN {X -0.026,Y -266.995,Z 488.259,A 0.000,B 0.000,C 90.000,E1 46.581} C_DIS
LIN {X 0.143,Y -260.311,Z 488.247,A 0.000,B 0.000,C 90.000,E1 44.433} C_DIS
LIN {X 0.041,Y -250.148,Z 488.229,A 0.000,B 0.000,C 90.000,E1 41.229} C_DIS
LIN {X 0.076,Y -240.441,Z 488.211,A 0.000,B 0.000,C 90.000,E1 37.935} C_DIS
LIN {X 0.014,Y -232.280,Z 488.194,A 0.000,B 0.000,C 90.000,E1 34.978} C_DIS
LIN {X 0.012,Y -224.944,Z 488.178,A 0.000,B 0.000,C 90.000,E1 31.957} C_DIS
LIN {X 0.084,Y -218.591,Z 488.161,A 0.000,B 0.000,C 90.000,E1 28.871} C_DIS
LIN {X -0.040,Y -213.000,Z 488.143,A 0.000,B 0.000,C 90.000,E1 25.796} C_DIS
LIN {X 0.022,Y -207.196,Z 488.121,A 0.000,B 0.000,C 90.000,E1 21.844} C_DIS
LIN {X -0.023,Y -202.411,Z 488.099,A 0.000,B 0.000,C 90.000,E1 17.873} C_DIS
LIN {X 0.054,Y -198.536,Z 488.077,A 0.000,B 0.000,C 90.000,E1 13.828} C_DIS
LIN {X 0.002,Y -195.337,Z 488.050,A 0.000,B 0.000,C 90.000,E1 8.973} C_DIS
LIN {X 0.035,Y -193.022,Z 488.009,A 0.000,B 0.000,C 90.000,E1 1.604} C_DIS
LIN {X -0.104,Y -194.825,Z 487.956,A 0.000,B 0.000,C 90.000,E1 352.186} C_DIS
LIN {X -0.079,Y -197.964,Z 487.929,A 0.000,B 0.000,C 90.000,E1 347.285} C_DIS
LIN {X -0.037,Y -202.438,Z 487.902,A 0.000,B 0.000,C 90.000,E1 342.417} C_DIS
LIN {X -0.046,Y -207.213,Z 487.880,A 0.000,B 0.000,C 90.000,E1 338.411} C_DIS
LIN {X 0.092,Y -212.726,Z 487.858,A 0.000,B 0.000,C 90.000,E1 334.409} C_DIS
LIN {X 0.019,Y -218.892,Z 487.836,A 0.000,B 0.000,C 90.000,E1 330.511} C_DIS
LIN {X 0.091,Y -225.627,Z 487.815,A 0.000,B 0.000,C 90.000,E1 326.628} C_DIS
LIN {X -0.013,Y -233.033,Z 487.794,A 0.000,B 0.000,C 90.000,E1 322.844} C_DIS
LIN {X -0.022,Y -241.262,Z 487.773,A 0.000,B 0.000,C 90.000,E1 319.094} C_DIS
LIN {X -0.004,Y -248.585,Z 487.756,A 0.000,B 0.000,C 90.000,E1 316.134} C_DIS
LIN {X 0.059,Y -257.941,Z 487.738,A 0.000,B 0.000,C 90.000,E1 312.852} C_DIS
LIN {X 0.144,Y -269.346,Z 487.718,A 0.000,B 0.000,C 90.000,E1 309.277} C_DIS
LIN {X 0.128,Y -282.054,Z 487.699,A 0.000,B 0.000,C 90.000,E1 305.804} C_DIS
LIN {X 0.092,Y -295.840,Z 487.680,A 0.000,B 0.000,C 90.000,E1 302.418} C_DIS
LIN {X -0.030,Y -309.066,Z 487.664,A 0.000,B 0.000,C 90.000,E1 299.461} C_DIS
LIN {X 0.035,Y -320.160,Z 487.651,A 0.000,B 0.000,C 90.000,E1 297.180} C_DIS
LIN {X -0.006,Y -336.077,Z 487.635,A 0.000,B 0.000,C 90.000,E1 294.335} C_DIS
LIN {X 0.128,Y -351.831,Z 487.621,A 0.000,B 0.000,C 90.000,E1 291.844} C_DIS
LIN {X 0.074,Y -369.227,Z 487.608,A 0.000,B 0.000,C 90.000,E1 289.450} C_DIS
LIN {X 0.084,Y -385.829,Z 487.597,A 0.000,B 0.000,C 90.000,E1 287.402} C_DIS
LIN {X -0.042,Y -410.812,Z 487.581,A 0.000,B 0.000,C 90.000,E1 284.592} C_DIS
LIN {X 0.121,Y -426.119,Z 487.572,A 0.000,B 0.000,C 90.000,E1 282.952} C_DIS
LIN {X -0.058,Y -438.480,Z 487.565,A 0.000,B 0.000,C 90.000,E1 281.658} C_DIS
LIN {X -0.054,Y -448.140,Z 487.559,A 0.000,B 0.000,C 90.000,E1 280.602} C_DIS
LIN {X 0.150,Y -454.888,Z 487.555,A 0.000,B 0.000,C 90.000,E1 279.792} C_DIS
LIN {X 0.037,Y -461.050,Z 487.550,A 0.000,B 0.000,C 90.000,E1 279.029} C_DIS
LIN {X 0.131,Y -468.398,Z 487.544,A 0.000,B 0.000,C 90.000,E1 277.992} C_DIS
LIN {X 0.065,Y -473.230,Z 487.540,A 0.000,B 0.000,C 90.000,E1 277.239} C_DIS
LIN {X 0.031,Y -477.526,Z 487.536,A 0.000,B 0.000,C 90.000,E1 276.486} C_DIS
LIN {X -0.017,Y -481.273,Z 487.532,A 0.000,B 0.000,C 90.000,E1 275.739} C_DIS
LIN {X -0.032,Y -484.413,Z 487.528,A 0.000,B 0.000,C 90.000,E1 274.992} C_DIS
LIN {X 0.145,Y -486.137,Z 487.525,A 0.000,B 0.000,C 90.000,E1 274.473} C_DIS
LIN {X -0.154,Y -487.546,Z 487.522,A 0.000,B 0.000,C 90.000,E1 274.012} C_DIS
LIN {X 0.009,Y -488.638,Z 487.519,A 0.000,B 0.000,C 90.000,E1 273.498} C_DIS
LIN {X 0.211,Y -489.422,Z 487.517,A 0.000,B 0.000,C 90.000,E1 272.980} C_DIS
LIN {X -0.095,Y -489.850,Z 487.514,A 0.000,B 0.000,C 90.000,E1 272.522} C_DIS
LIN {X 0.095,Y -489.911,Z 487.511,A 0.000,B 0.000,C 90.000,E1 272.007} C_DIS
LIN {X -0.186,Y -489.544,Z 487.508,A 0.000,B 0.000,C 90.000,E1 271.547} C_DIS
LIN {X 0.006,Y -488.721,Z 487.506,A 0.000,B 0.000,C 90.000,E1 271.031} C_DIS
LIN {X 0.198,Y -487.424,Z 487.503,A 0.000,B 0.000,C 90.000,E1 270.516} C_DIS
LIN {X -0.102,Y -485.532,Z 487.500,A 0.000,B 0.000,C 90.000,E1 270.057} C_DIS
LIN {X 0.079,Y -482.961,Z 487.497,A 0.000,B 0.000,C 90.000,E1 269.542} C_DIS
LIN {X 0.237,Y -479.672,Z 487.495,A 0.000,B 0.000,C 90.000,E1 269.026} C_DIS
LIN {X -0.099,Y -475.414,Z 487.492,A 0.000,B 0.000,C 90.000,E1 268.568} C_DIS
LIN {X 0.034,Y -470.169,Z 487.489,A 0.000,B 0.000,C 90.000,E1 268.051} C_DIS
LIN {X -0.029,Y -464.139,Z 487.487,A 0.000,B 0.000,C 90.000,E1 267.593} C_DIS
LIN {X -0.069,Y -457.541,Z 487.484,A 0.000,B 0.000,C 90.000,E1 267.192} C_DIS
LIN {X -0.014,Y -450.573,Z 487.482,A 0.000,B 0.000,C 90.000,E1 266.846} C_DIS
LIN {X 0.053,Y -443.724,Z 487.481,A 0.000,B 0.000,C 90.000,E1 266.560} C_DIS
LIN {X -0.003,Y -436.218,Z 487.480,A 0.000,B 0.000,C 90.000,E1 266.331} C_DIS
LIN {X -0.099,Y -427.707,Z 487.479,A 0.000,B 0.000,C 90.000,E1 266.159} C_DIS
LIN {X -0.183,Y -418.615,Z 487.478,A 0.000,B 0.000,C 90.000,E1 266.045} C_DIS
LIN {X -0.161,Y -411.111,Z 487.478,A 0.000,B 0.000,C 90.000,E1 265.988} C_DIS
LIN {X 0.168,Y -406.084,Z 487.478,A 0.000,B 0.000,C 90.000,E1 265.931} C_DIS
LIN {X 0.053,Y -180.918,Z 487.477,A 0.000,B 0.000,C 90.000,E1 265.927} C_DIS
LIN {X 0.082,Y -180.841,Z 487.472,A 0.000,B 0.000,C 90.000,E1 264.894} C_DIS
LIN {X -0.022,Y -178.884,Z 487.443,A 0.000,B 0.000,C 90.000,E1 259.690} C_DIS
LIN {X 0.054,Y -175.926,Z 487.414,A 0.000,B 0.000,C 90.000,E1 254.574} C_DIS
LIN {X 0.000,Y -175.368,Z 487.410,A 0.000,B 0.000,C 90.000,E1 253.740} C_DIS
LIN {X 0.058,Y -172.145,Z 487.386,A 0.000,B 0.000,C 90.000,E1 249.444} C_DIS
LIN {X 0.035,Y -171.609,Z 487.381,A 0.000,B 0.000,C 90.000,E1 248.592} C_DIS
LIN {X 0.024,Y -167.832,Z 487.357,A 0.000,B 0.000,C 90.000,E1 244.280} C_DIS
LIN {X 0.041,Y -166.558,Z 487.348,A 0.000,B 0.000,C 90.000,E1 242.538} C_DIS
LIN {X -0.049,Y -162.553,Z 487.323,A 0.000,B 0.000,C 90.000,E1 238.201} C_DIS
LIN {X 0.011,Y -161.231,Z 487.313,A 0.000,B 0.000,C 90.000,E1 236.421} C_DIS
LIN {X 0.046,Y -157.237,Z 487.289,A 0.000,B 0.000,C 90.000,E1 231.984} C_DIS
LIN {X -0.031,Y -155.961,Z 487.279,A 0.000,B 0.000,C 90.000,E1 230.231} C_DIS
LIN {X 0.027,Y -152.215,Z 487.254,A 0.000,B 0.000,C 90.000,E1 225.729} C_DIS
LIN {X 0.048,Y -150.459,Z 487.239,A 0.000,B 0.000,C 90.000,E1 223.014} C_DIS
LIN {X 0.074,Y -147.185,Z 487.214,A 0.000,B 0.000,C 90.000,E1 218.463} C_DIS
LIN {X 0.040,Y -145.202,Z 487.194,A 0.000,B 0.000,C 90.000,E1 214.818} C_DIS
LIN {X -0.050,Y -142.339,Z 487.163,A 0.000,B 0.000,C 90.000,E1 209.333} C_DIS
LIN {X 0.004,Y -141.727,Z 487.153,A 0.000,B 0.000,C 90.000,E1 207.462} C_DIS
LIN {X -0.014,Y -139.481,Z 487.116,A 0.000,B 0.000,C 90.000,E1 200.972} C_DIS
LIN {X -0.025,Y -138.979,Z 487.101,A 0.000,B 0.000,C 90.000,E1 198.181} C_DIS
LIN {X -0.040,Y -138.333,Z 487.054,A 0.000,B 0.000,C 90.000,E1 189.782} C_DIS
LIN {X -0.040,Y -139.429,Z 487.008,A 0.000,B 0.000,C 90.000,E1 181.375} C_DIS
LIN {X 0.013,Y -141.356,Z 486.971,A 0.000,B 0.000,C 90.000,E1 174.837} C_DIS
LIN {X -0.010,Y -142.710,Z 486.956,A 0.000,B 0.000,C 90.000,E1 172.064} C_DIS
LIN {X -0.052,Y -145.084,Z 486.930,A 0.000,B 0.000,C 90.000,E1 167.465} C_DIS
LIN {X -0.056,Y -147.708,Z 486.910,A 0.000,B 0.000,C 90.000,E1 163.795} C_DIS
LIN {X 0.028,Y -150.364,Z 486.890,A 0.000,B 0.000,C 90.000,E1 160.115} C_DIS
LIN {X 0.046,Y -153.789,Z 486.869,A 0.000,B 0.000,C 90.000,E1 156.485} C_DIS
LIN {X -0.034,Y -157.201,Z 486.849,A 0.000,B 0.000,C 90.000,E1 152.922} C_DIS
LIN {X 0.048,Y -161.364,Z 486.830,A 0.000,B 0.000,C 90.000,E1 149.331} C_DIS
LIN {X 0.059,Y -165.566,Z 486.810,A 0.000,B 0.000,C 90.000,E1 145.801} C_DIS
LIN {X -0.057,Y -170.484,Z 486.791,A 0.000,B 0.000,C 90.000,E1 142.351} C_DIS
LIN {X 0.092,Y -175.365,Z 486.772,A 0.000,B 0.000,C 90.000,E1 138.852} C_DIS
LIN {X -0.045,Y -180.989,Z 486.753,A 0.000,B 0.000,C 90.000,E1 135.486} C_DIS
LIN {X 0.080,Y -186.416,Z 486.734,A 0.000,B 0.000,C 90.000,E1 132.081} C_DIS
LIN {X -0.120,Y -191.042,Z 486.720,A 0.000,B 0.000,C 90.000,E1 129.644} C_DIS
LIN {X -0.070,Y -193.331,Z 486.712,A 0.000,B 0.000,C 90.000,E1 128.257} C_DIS
LIN {X 0.023,Y -290.772,Z 486.712,A 0.000,B 0.000,C 90.000,E1 128.222} C_DIS
LIN {X -0.021,Y -295.161,Z 486.712,A 0.000,B 0.000,C 90.000,E1 128.096} C_DIS
LIN {X -0.065,Y -297.259,Z 486.711,A 0.000,B 0.000,C 90.000,E1 127.971} C_DIS
LIN {X 0.006,Y -301.135,Z 486.709,A 0.000,B 0.000,C 90.000,E1 127.569} C_DIS
LIN {X 0.032,Y -304.642,Z 486.706,A 0.000,B 0.000,C 90.000,E1 126.996} C_DIS
LIN {X 0.043,Y -306.082,Z 486.704,A 0.000,B 0.000,C 90.000,E1 126.664} C_DIS
LIN {X -0.191,Y -307.219,Z 486.702,A 0.000,B 0.000,C 90.000,E1 126.377} C_DIS
LIN {X 0.020,Y -317.328,Z 486.684,A 0.000,B 0.000,C 90.000,E1 123.086} C_DIS
LIN {X 0.057,Y -327.745,Z 486.668,A 0.000,B 0.000,C 90.000,E1 120.207} C_DIS
LIN {X 0.067,Y -339.524,Z 486.652,A 0.000,B 0.000,C 90.000,E1 117.385} C_DIS
LIN {X -0.058,Y -352.766,Z 486.637,A 0.000,B 0.000,C 90.000,E1 114.643} C_DIS
LIN {X 0.153,Y -365.865,Z 486.624,A 0.000,B 0.000,C 90.000,E1 112.206} C_DIS
LIN {X -0.052,Y -380.313,Z 486.610,A 0.000,B 0.000,C 90.000,E1 109.885} C_DIS
LIN {X -0.025,Y -396.214,Z 486.598,A 0.000,B 0.000,C 90.000,E1 107.583} C_DIS
LIN {X -0.229,Y -413.685,Z 486.585,A 0.000,B 0.000,C 90.000,E1 105.371} C_DIS
LIN {X -0.108,Y -432.832,Z 486.573,A 0.000,B 0.000,C 90.000,E1 103.175} C_DIS
END
